Yaskawa INFORM job: DEMO_ROOF_UPPER_0625_3PAINT_33.JBI

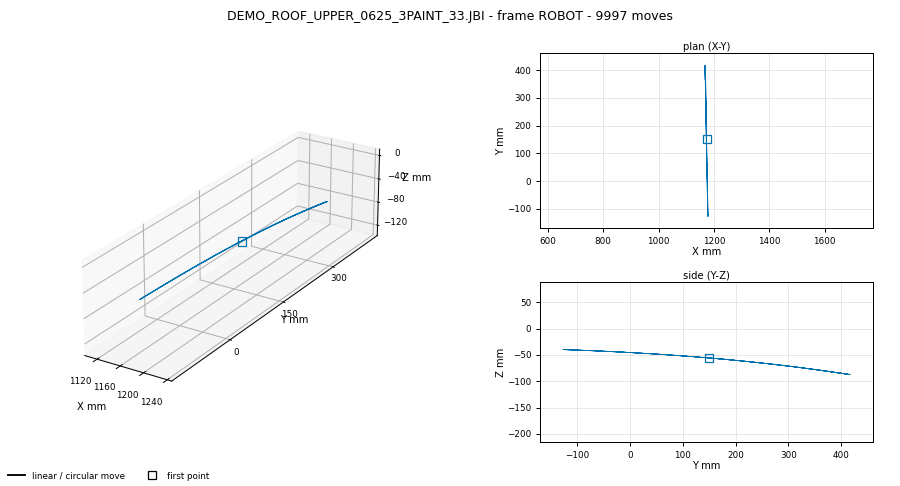
[picture p0: tool path of DEMO_ROOF_UPPER_0625_3PAINT_33.JBI in frame ROBOT, 9997 of 9997 moves have a stored position in this frame; points joined in program order, loops and branches not executed]
/JOB
//NAME DEMO_ROOF_UPPER_0625_3PAINT33
//POS
///NPOS 9997,0,0,0,0,0
///TOOL 0
///USER 0
///POSTYPE ROBOT
///RECTAN
///RCONF 1,0,0,0,0,0,0,0,0,0,0,0,0,0,0,0,0,0,0,0,0,0,0,0
C00000=1173.665,150.338,-55.820,-178.432,6.530,148.733
C00001=1173.661,150.587,-55.840,-178.430,6.532,148.732
C00002=1173.656,150.836,-55.861,-178.427,6.533,148.732
C00003=1173.651,151.085,-55.883,-178.424,6.535,148.732
C00004=1173.646,151.335,-55.904,-178.422,6.536,148.731
C00005=1173.642,151.583,-55.925,-178.420,6.538,148.731
C00006=1173.637,151.832,-55.946,-178.417,6.540,148.730
C00007=1173.632,152.082,-55.967,-178.414,6.541,148.730
C00008=1173.627,152.330,-55.988,-178.411,6.543,148.730
C00009=1173.623,152.580,-56.010,-178.409,6.545,148.729
C00010=1173.618,152.828,-56.031,-178.406,6.547,148.729
C00011=1173.613,153.078,-56.052,-178.403,6.548,148.728
C00012=1173.608,153.327,-56.073,-178.401,6.550,148.728
C00013=1173.604,153.575,-56.094,-178.398,6.552,148.728
C00014=1173.599,153.825,-56.116,-178.395,6.554,148.727
C00015=1173.594,154.074,-56.137,-178.393,6.555,148.727
C00016=1173.590,154.323,-56.158,-178.390,6.557,148.727
C00017=1173.585,154.571,-56.179,-178.387,6.559,148.726
C00018=1173.580,154.821,-56.201,-178.385,6.561,148.726
C00019=1173.575,155.070,-56.223,-178.382,6.562,148.725
C00020=1173.571,155.319,-56.243,-178.379,6.564,148.725
C00021=1173.566,155.568,-56.265,-178.377,6.566,148.725
C00022=1173.562,155.817,-56.287,-178.374,6.568,148.724
C00023=1173.557,156.066,-56.308,-178.371,6.570,148.724
C00024=1173.552,156.315,-56.329,-178.368,6.571,148.724
C00025=1173.547,156.564,-56.350,-178.366,6.573,148.723
C00026=1173.543,156.813,-56.372,-178.363,6.575,148.723
C00027=1173.538,157.062,-56.393,-178.360,6.577,148.722
C00028=1173.533,157.311,-56.414,-178.358,6.578,148.722
C00029=1173.529,157.560,-56.436,-178.355,6.580,148.721
C00030=1173.524,157.810,-56.457,-178.352,6.581,148.721
C00031=1173.519,158.078,-56.481,-178.349,6.583,148.721
C00032=1173.514,158.348,-56.504,-178.346,6.586,148.720
C00033=1173.509,158.617,-56.527,-178.343,6.588,148.720
C00034=1173.504,158.885,-56.551,-178.340,6.589,148.720
C00035=1173.499,159.135,-56.572,-178.338,6.591,148.719
C00036=1173.494,159.383,-56.594,-178.335,6.593,148.719
C00037=1173.489,159.633,-56.616,-178.332,6.595,148.719
C00038=1173.484,159.882,-56.637,-178.330,6.596,148.718
C00039=1173.480,160.130,-56.658,-178.327,6.598,148.718
C00040=1173.476,160.379,-56.680,-178.324,6.600,148.717
C00041=1173.471,160.628,-56.701,-178.322,6.602,148.717
C00042=1173.466,160.877,-56.723,-178.319,6.603,148.717
C00043=1173.462,161.127,-56.745,-178.316,6.605,148.716
C00044=1173.457,161.375,-56.766,-178.314,6.607,148.716
C00045=1173.452,161.625,-56.788,-178.311,6.609,148.716
C00046=1173.448,161.873,-56.810,-178.308,6.610,148.715
C00047=1173.443,162.122,-56.832,-178.306,6.612,148.715
C00048=1173.438,162.371,-56.854,-178.303,6.614,148.714
C00049=1173.433,162.621,-56.875,-178.300,6.616,148.714
C00050=1173.429,162.870,-56.897,-178.297,6.618,148.714
C00051=1173.424,163.119,-56.918,-178.294,6.620,148.713
C00052=1173.419,163.367,-56.940,-178.292,6.622,148.713
C00053=1173.415,163.617,-56.962,-178.289,6.624,148.713
C00054=1173.410,163.865,-56.984,-178.286,6.625,148.712
C00055=1173.405,164.115,-57.006,-178.283,6.627,148.712
C00056=1173.400,164.363,-57.028,-178.281,6.629,148.711
C00057=1173.396,164.613,-57.050,-178.278,6.631,148.711
C00058=1173.391,164.861,-57.072,-178.275,6.632,148.711
C00059=1173.386,165.110,-57.094,-178.273,6.634,148.710
C00060=1173.382,165.359,-57.116,-178.271,6.636,148.710
C00061=1173.377,165.608,-57.137,-178.268,6.638,148.710
C00062=1173.373,165.857,-57.159,-178.265,6.640,148.709
C00063=1173.368,166.106,-57.181,-178.262,6.641,148.709
C00064=1173.364,166.355,-57.203,-178.260,6.643,148.709
C00065=1173.358,166.604,-57.225,-178.257,6.645,148.708
C00066=1173.354,166.854,-57.247,-178.254,6.647,148.708
C00067=1173.349,167.102,-57.269,-178.251,6.649,148.708
C00068=1173.345,167.352,-57.291,-178.248,6.651,148.707
C00069=1173.340,167.600,-57.313,-178.246,6.653,148.707
C00070=1173.335,167.850,-57.335,-178.243,6.655,148.707
C00071=1173.330,168.099,-57.357,-178.240,6.656,148.706
C00072=1173.326,168.348,-57.379,-178.238,6.658,148.706
C00073=1173.321,168.597,-57.401,-178.235,6.660,148.705
C00074=1173.317,168.845,-57.424,-178.232,6.662,148.705
C00075=1173.312,169.094,-57.445,-178.230,6.663,148.705
C00076=1173.307,169.344,-57.468,-178.227,6.666,148.705
C00077=1173.302,169.592,-57.490,-178.225,6.667,148.704
C00078=1173.298,169.842,-57.512,-178.222,6.669,148.704
C00079=1173.293,170.090,-57.534,-178.219,6.671,148.703
C00080=1173.288,170.339,-57.557,-178.216,6.673,148.703
C00081=1173.283,170.588,-57.578,-178.213,6.675,148.703
C00082=1173.279,170.837,-57.600,-178.211,6.677,148.702
C00083=1173.275,171.087,-57.622,-178.208,6.679,148.702
C00084=1173.269,171.335,-57.645,-178.205,6.680,148.702
C00085=1173.265,171.584,-57.667,-178.203,6.682,148.701
C00086=1173.260,171.833,-57.689,-178.200,6.684,148.701
C00087=1173.256,172.082,-57.713,-178.197,6.686,148.701
C00088=1173.251,172.331,-57.734,-178.195,6.688,148.700
C00089=1173.247,172.580,-57.756,-178.192,6.690,148.700
C00090=1173.241,172.830,-57.779,-178.189,6.692,148.700
C00091=1173.237,173.078,-57.801,-178.187,6.694,148.699
C00092=1173.233,173.327,-57.823,-178.184,6.696,148.699
C00093=1173.227,173.575,-57.846,-178.181,6.698,148.699
C00094=1173.223,173.825,-57.868,-178.178,6.699,148.698
C00095=1173.219,174.074,-57.890,-178.176,6.701,148.698
C00096=1173.214,174.322,-57.913,-178.173,6.703,148.698
C00097=1173.209,174.572,-57.935,-178.171,6.705,148.697
C00098=1173.205,174.821,-57.958,-178.168,6.708,148.697
C00099=1173.200,175.069,-57.981,-178.165,6.709,148.697
C00100=1173.195,175.319,-58.003,-178.162,6.711,148.696
C00101=1173.190,175.567,-58.026,-178.160,6.713,148.696
C00102=1173.186,175.816,-58.048,-178.157,6.715,148.696
C00103=1173.181,176.065,-58.071,-178.154,6.716,148.695
C00104=1173.176,176.314,-58.093,-178.152,6.718,148.695
C00105=1173.172,176.563,-58.115,-178.149,6.721,148.695
C00106=1173.167,176.812,-58.138,-178.146,6.723,148.694
C00107=1173.163,177.060,-58.160,-178.143,6.725,148.694
C00108=1173.158,177.310,-58.183,-178.141,6.726,148.694
C00109=1173.154,177.559,-58.206,-178.138,6.728,148.693
C00110=1173.149,177.808,-58.229,-178.135,6.730,148.693
C00111=1173.144,178.056,-58.251,-178.133,6.732,148.693
C00112=1173.140,178.305,-58.274,-178.130,6.735,148.692
C00113=1173.135,178.555,-58.296,-178.127,6.736,148.692
C00114=1173.130,178.803,-58.319,-178.125,6.738,148.692
C00115=1173.126,179.052,-58.341,-178.122,6.740,148.691
C00116=1173.121,179.301,-58.365,-178.119,6.742,148.691
C00117=1173.117,179.550,-58.387,-178.117,6.743,148.691
C00118=1173.111,179.799,-58.410,-178.114,6.745,148.690
C00119=1173.107,180.048,-58.433,-178.111,6.748,148.690
C00120=1173.103,180.297,-58.456,-178.108,6.750,148.690
C00121=1173.098,180.546,-58.478,-178.106,6.752,148.689
C00122=1173.093,180.795,-58.501,-178.103,6.753,148.689
C00123=1173.088,181.044,-58.524,-178.100,6.755,148.689
C00124=1173.084,181.293,-58.546,-178.098,6.757,148.688
C00125=1173.080,181.542,-58.570,-178.095,6.760,148.688
C00126=1173.075,181.790,-58.592,-178.092,6.762,148.688
C00127=1173.070,182.039,-58.615,-178.090,6.764,148.688
C00128=1173.065,182.289,-58.638,-178.087,6.765,148.687
C00129=1173.061,182.537,-58.661,-178.084,6.767,148.687
C00130=1173.056,182.786,-58.684,-178.081,6.770,148.686
C00131=1173.051,183.035,-58.707,-178.079,6.772,148.686
C00132=1173.047,183.284,-58.729,-178.076,6.774,148.686
C00133=1173.042,183.533,-58.753,-178.073,6.775,148.686
C00134=1173.038,183.782,-58.775,-178.071,6.777,148.685
C00135=1173.033,184.052,-58.800,-178.067,6.780,148.685
C00136=1173.028,184.321,-58.825,-178.065,6.781,148.685
C00137=1173.023,184.591,-58.850,-178.062,6.784,148.684
C00138=1173.018,184.860,-58.876,-178.059,6.786,148.684
C00139=1173.013,185.110,-58.898,-178.056,6.788,148.684
C00140=1173.009,185.358,-58.921,-178.053,6.791,148.683
C00141=1173.004,185.607,-58.944,-178.051,6.792,148.683
C00142=1172.999,185.856,-58.967,-178.048,6.794,148.683
C00143=1172.994,186.105,-58.991,-178.045,6.796,148.682
C00144=1172.990,186.353,-59.014,-178.043,6.798,148.682
C00145=1172.986,186.603,-59.037,-178.040,6.801,148.682
C00146=1172.981,186.852,-59.060,-178.037,6.802,148.681
C00147=1172.976,187.101,-59.084,-178.035,6.804,148.681
C00148=1172.972,187.349,-59.106,-178.032,6.806,148.681
C00149=1172.967,187.598,-59.129,-178.030,6.808,148.681
C00150=1172.962,187.847,-59.153,-178.026,6.811,148.680
C00151=1172.958,188.096,-59.176,-178.024,6.812,148.680
C00152=1172.953,188.345,-59.199,-178.021,6.814,148.680
C00153=1172.949,188.593,-59.222,-178.018,6.816,148.679
C00154=1172.944,188.842,-59.246,-178.016,6.819,148.679
C00155=1172.940,189.092,-59.269,-178.013,6.821,148.679
C00156=1172.935,189.341,-59.292,-178.010,6.822,148.678
C00157=1172.930,189.589,-59.315,-178.008,6.824,148.678
C00158=1172.925,189.837,-59.339,-178.005,6.826,148.678
C00159=1172.921,190.086,-59.363,-178.002,6.829,148.678
C00160=1172.917,190.335,-59.385,-177.999,6.831,148.677
C00161=1172.912,190.584,-59.409,-177.997,6.832,148.677
C00162=1172.907,190.833,-59.432,-177.995,6.835,148.677
C00163=1172.903,191.082,-59.456,-177.991,6.837,148.676
C00164=1172.898,191.331,-59.479,-177.989,6.839,148.676
C00165=1172.893,191.580,-59.503,-177.986,6.841,148.676
C00166=1172.889,191.829,-59.526,-177.983,6.842,148.675
C00167=1172.884,192.078,-59.550,-177.981,6.845,148.675
C00168=1172.879,192.327,-59.573,-177.978,6.847,148.675
C00169=1172.875,192.575,-59.597,-177.975,6.849,148.675
C00170=1172.870,192.824,-59.620,-177.973,6.851,148.674
C00171=1172.866,193.073,-59.644,-177.970,6.854,148.674
C00172=1172.861,193.322,-59.667,-177.967,6.855,148.674
C00173=1172.856,193.571,-59.691,-177.964,6.857,148.673
C00174=1172.852,193.820,-59.715,-177.962,6.859,148.673
C00175=1172.847,194.069,-59.738,-177.959,6.862,148.673
C00176=1172.843,194.317,-59.762,-177.956,6.864,148.673
C00177=1172.838,194.566,-59.785,-177.954,6.866,148.672
C00178=1172.833,194.815,-59.809,-177.951,6.868,148.672
C00179=1172.829,195.064,-59.833,-177.948,6.870,148.672
C00180=1172.824,195.313,-59.856,-177.946,6.872,148.671
C00181=1172.819,195.562,-59.880,-177.943,6.874,148.671
C00182=1172.815,195.810,-59.904,-177.940,6.877,148.671
C00183=1172.810,196.059,-59.927,-177.937,6.879,148.671
C00184=1172.806,196.307,-59.951,-177.935,6.880,148.670
C00185=1172.801,196.557,-59.974,-177.933,6.882,148.670
C00186=1172.797,196.806,-59.998,-177.929,6.885,148.670
C00187=1172.792,197.054,-60.022,-177.927,6.887,148.669
C00188=1172.787,197.303,-60.045,-177.924,6.889,148.669
C00189=1172.784,197.552,-60.070,-177.921,6.892,148.669
C00190=1172.779,197.801,-60.093,-177.918,6.893,148.669
C00191=1172.775,198.050,-60.117,-177.916,6.895,148.668
C00192=1172.769,198.299,-60.141,-177.914,6.897,148.668
C00193=1172.765,198.547,-60.165,-177.910,6.900,148.668
C00194=1172.760,198.796,-60.188,-177.908,6.902,148.668
C00195=1172.756,199.045,-60.213,-177.905,6.903,148.667
C00196=1172.751,199.294,-60.236,-177.902,6.906,148.667
C00197=1172.747,199.542,-60.260,-177.900,6.908,148.667
C00198=1172.742,199.791,-60.284,-177.897,6.910,148.666
C00199=1172.737,200.041,-60.308,-177.894,6.913,148.666
C00200=1172.733,200.289,-60.332,-177.891,6.915,148.666
C00201=1172.728,200.538,-60.356,-177.889,6.916,148.666
C00202=1172.724,200.787,-60.380,-177.887,6.919,148.665
C00203=1172.719,201.035,-60.404,-177.883,6.921,148.665
C00204=1172.714,201.284,-60.428,-177.881,6.923,148.665
C00205=1172.710,201.533,-60.452,-177.879,6.925,148.665
C00206=1172.706,201.782,-60.476,-177.875,6.928,148.664
C00207=1172.701,202.031,-60.500,-177.873,6.929,148.664
C00208=1172.697,202.279,-60.524,-177.870,6.932,148.664
C00209=1172.692,202.528,-60.549,-177.867,6.934,148.664
C00210=1172.687,202.776,-60.573,-177.864,6.936,148.663
C00211=1172.683,203.026,-60.596,-177.862,6.938,148.663
C00212=1172.678,203.275,-60.621,-177.859,6.941,148.663
C00213=1172.674,203.523,-60.645,-177.856,6.942,148.662
C00214=1172.669,203.772,-60.669,-177.854,6.945,148.662
C00215=1172.664,204.021,-60.693,-177.851,6.947,148.662
C00216=1172.660,204.270,-60.718,-177.848,6.949,148.662
C00217=1172.656,204.519,-60.742,-177.846,6.951,148.662
C00218=1172.651,204.767,-60.766,-177.843,6.954,148.661
C00219=1172.646,205.016,-60.790,-177.840,6.955,148.661
C00220=1172.642,205.265,-60.814,-177.838,6.958,148.661
C00221=1172.638,205.514,-60.838,-177.835,6.960,148.660
C00222=1172.632,205.763,-60.863,-177.832,6.962,148.660
C00223=1172.628,206.011,-60.887,-177.830,6.964,148.660
C00224=1172.623,206.260,-60.912,-177.827,6.967,148.660
C00225=1172.619,206.509,-60.936,-177.824,6.969,148.660
C00226=1172.615,206.757,-60.960,-177.822,6.971,148.659
C00227=1172.610,207.006,-60.985,-177.819,6.973,148.659
C00228=1172.606,207.255,-61.009,-177.816,6.975,148.659
C00229=1172.601,207.504,-61.034,-177.813,6.978,148.658
C00230=1172.596,207.753,-61.057,-177.810,6.980,148.658
C00231=1172.592,208.001,-61.081,-177.808,6.982,148.658
C00232=1172.587,208.251,-61.106,-177.805,6.984,148.658
C00233=1172.583,208.499,-61.130,-177.803,6.987,148.658
C00234=1172.577,208.748,-61.155,-177.800,6.988,148.657
C00235=1172.574,208.997,-61.180,-177.797,6.991,148.657
C00236=1172.569,209.246,-61.204,-177.795,6.993,148.657
C00237=1172.564,209.493,-61.229,-177.792,6.995,148.656
C00238=1172.559,209.742,-61.254,-177.789,6.998,148.656
C00239=1172.554,210.014,-61.280,-177.786,7.000,148.656
C00240=1172.549,210.284,-61.307,-177.783,7.002,148.656
C00241=1172.545,210.554,-61.333,-177.780,7.005,148.655
C00242=1172.540,210.824,-61.360,-177.777,7.007,148.655
C00243=1172.535,211.073,-61.385,-177.775,7.010,148.655
C00244=1172.531,211.322,-61.409,-177.772,7.011,148.655
C00245=1172.526,211.571,-61.434,-177.769,7.014,148.654
C00246=1172.521,211.819,-61.459,-177.767,7.016,148.654
C00247=1172.518,212.068,-61.484,-177.764,7.018,148.654
C00248=1172.513,212.317,-61.508,-177.761,7.021,148.654
C00249=1172.508,212.565,-61.532,-177.759,7.023,148.653
C00250=1172.504,212.815,-61.557,-177.756,7.026,148.653
C00251=1172.500,213.063,-61.582,-177.753,7.027,148.653
C00252=1172.495,213.312,-61.607,-177.751,7.029,148.653
C00253=1172.490,213.561,-61.632,-177.748,7.032,148.652
C00254=1172.485,213.809,-61.656,-177.745,7.034,148.652
C00255=1172.481,214.058,-61.682,-177.742,7.037,148.652
C00256=1172.476,214.307,-61.706,-177.740,7.039,148.652
C00257=1172.472,214.556,-61.731,-177.737,7.042,148.652
C00258=1172.467,214.805,-61.755,-177.734,7.043,148.651
C00259=1172.463,215.052,-61.780,-177.732,7.046,148.651
C00260=1172.459,215.302,-61.805,-177.729,7.048,148.651
C00261=1172.453,215.550,-61.830,-177.726,7.050,148.651
C00262=1172.449,215.799,-61.856,-177.723,7.053,148.650
C00263=1172.445,216.048,-61.880,-177.721,7.055,148.650
C00264=1172.441,216.297,-61.905,-177.718,7.057,148.650
C00265=1172.435,216.545,-61.930,-177.715,7.059,148.650
C00266=1172.432,216.794,-61.955,-177.713,7.062,148.650
C00267=1172.427,217.042,-61.980,-177.710,7.064,148.649
C00268=1172.422,217.292,-62.005,-177.708,7.066,148.649
C00269=1172.418,217.540,-62.030,-177.704,7.069,148.649
C00270=1172.414,217.789,-62.055,-177.702,7.071,148.648
C00271=1172.409,218.038,-62.080,-177.700,7.073,148.648
C00272=1172.404,218.287,-62.105,-177.696,7.075,148.648
C00273=1172.400,218.535,-62.129,-177.694,7.078,148.648
C00274=1172.396,218.784,-62.155,-177.691,7.080,148.648
C00275=1172.391,219.033,-62.180,-177.689,7.082,148.648
C00276=1172.386,219.281,-62.206,-177.685,7.085,148.647
C00277=1172.382,219.529,-62.231,-177.683,7.087,148.647
C00278=1172.378,219.779,-62.255,-177.680,7.090,148.647
C00279=1172.373,220.027,-62.281,-177.678,7.092,148.647
C00280=1172.368,220.276,-62.306,-177.675,7.094,148.646
C00281=1172.364,220.524,-62.331,-177.672,7.097,148.646
C00282=1172.359,220.774,-62.356,-177.670,7.098,148.646
C00283=1172.354,221.022,-62.382,-177.667,7.101,148.646
C00284=1172.351,221.270,-62.407,-177.664,7.103,148.646
C00285=1172.346,221.519,-62.431,-177.662,7.106,148.645
C00286=1172.341,221.768,-62.457,-177.659,7.108,148.645
C00287=1172.337,222.017,-62.483,-177.656,7.111,148.645
C00288=1172.332,222.265,-62.508,-177.653,7.113,148.645
C00289=1172.328,222.514,-62.533,-177.651,7.115,148.645
C00290=1172.323,222.762,-62.559,-177.648,7.117,148.644
C00291=1172.318,223.012,-62.584,-177.645,7.120,148.644
C00292=1172.314,223.260,-62.609,-177.643,7.122,148.644
C00293=1172.309,223.509,-62.635,-177.640,7.124,148.644
C00294=1172.306,223.758,-62.659,-177.637,7.127,148.643
C00295=1172.301,224.006,-62.685,-177.635,7.129,148.643
C00296=1172.297,224.255,-62.710,-177.632,7.132,148.643
C00297=1172.292,224.503,-62.736,-177.630,7.134,148.643
C00298=1172.288,224.751,-62.762,-177.626,7.136,148.643
C00299=1172.283,225.001,-62.787,-177.624,7.138,148.642
C00300=1172.278,225.249,-62.812,-177.621,7.141,148.642
C00301=1172.274,225.498,-62.838,-177.619,7.143,148.642
C00302=1172.270,225.747,-62.863,-177.616,7.146,148.642
C00303=1172.265,225.995,-62.889,-177.613,7.148,148.642
C00304=1172.261,226.244,-62.915,-177.610,7.151,148.641
C00305=1172.256,226.493,-62.940,-177.608,7.153,148.641
C00306=1172.251,226.741,-62.965,-177.605,7.155,148.641
C00307=1172.247,226.990,-62.991,-177.603,7.157,148.641
C00308=1172.243,227.239,-63.017,-177.599,7.160,148.641
C00309=1172.237,227.487,-63.043,-177.597,7.162,148.640
C00310=1172.233,227.736,-63.068,-177.594,7.165,148.640
C00311=1172.229,227.985,-63.094,-177.592,7.167,148.640
C00312=1172.224,228.233,-63.119,-177.589,7.170,148.640
C00313=1172.220,228.482,-63.145,-177.586,7.172,148.640
C00314=1172.216,228.730,-63.171,-177.584,7.175,148.640
C00315=1172.211,228.978,-63.196,-177.581,7.176,148.639
C00316=1172.206,229.227,-63.222,-177.578,7.179,148.639
C00317=1172.202,229.476,-63.248,-177.576,7.182,148.639
C00318=1172.198,229.725,-63.274,-177.573,7.184,148.639
C00319=1172.192,229.973,-63.300,-177.570,7.186,148.639
C00320=1172.188,230.222,-63.325,-177.567,7.189,148.638
C00321=1172.184,230.471,-63.351,-177.565,7.192,148.638
C00322=1172.180,230.720,-63.377,-177.562,7.194,148.638
C00323=1172.175,230.968,-63.402,-177.559,7.197,148.638
C00324=1172.171,231.217,-63.428,-177.557,7.199,148.638
C00325=1172.166,231.465,-63.455,-177.554,7.201,148.637
C00326=1172.162,231.714,-63.481,-177.551,7.203,148.637
C00327=1172.157,231.962,-63.506,-177.548,7.206,148.637
C00328=1172.153,232.211,-63.532,-177.546,7.208,148.637
C00329=1172.149,232.460,-63.558,-177.543,7.211,148.637
C00330=1172.144,232.709,-63.584,-177.541,7.213,148.637
C00331=1172.139,232.958,-63.610,-177.538,7.216,148.636
C00332=1172.135,233.205,-63.636,-177.535,7.218,148.636
C00333=1172.131,233.454,-63.662,-177.533,7.221,148.636
C00334=1172.126,233.703,-63.688,-177.530,7.224,148.636
C00335=1172.121,233.952,-63.714,-177.527,7.225,148.636
C00336=1172.118,234.200,-63.740,-177.524,7.228,148.636
C00337=1172.112,234.448,-63.766,-177.522,7.230,148.635
C00338=1172.108,234.697,-63.792,-177.519,7.233,148.635
C00339=1172.104,234.945,-63.818,-177.517,7.235,148.635
C00340=1172.100,235.194,-63.844,-177.514,7.238,148.635
C00341=1172.095,235.443,-63.870,-177.511,7.240,148.635
C00342=1172.090,235.692,-63.896,-177.509,7.243,148.635
C00343=1172.085,235.963,-63.925,-177.505,7.246,148.634
C00344=1172.080,236.234,-63.954,-177.503,7.249,148.634
C00345=1172.076,236.506,-63.982,-177.499,7.251,148.634
C00346=1172.071,236.778,-64.011,-177.497,7.254,148.634
C00347=1172.066,237.027,-64.037,-177.494,7.256,148.634
C00348=1172.062,237.275,-64.063,-177.491,7.259,148.633
C00349=1172.057,237.524,-64.090,-177.489,7.261,148.633
C00350=1172.053,237.773,-64.116,-177.486,7.264,148.633
C00351=1172.049,238.021,-64.142,-177.484,7.266,148.633
C00352=1172.044,238.269,-64.168,-177.480,7.268,148.633
C00353=1172.040,238.517,-64.195,-177.478,7.271,148.633
C00354=1172.035,238.767,-64.221,-177.475,7.274,148.632
C00355=1172.031,239.015,-64.247,-177.472,7.276,148.632
C00356=1172.026,239.264,-64.274,-177.470,7.278,148.632
C00357=1172.022,239.512,-64.300,-177.467,7.281,148.632
C00358=1172.017,239.761,-64.327,-177.464,7.284,148.632
C00359=1172.013,240.009,-64.353,-177.462,7.286,148.632
C00360=1172.008,240.258,-64.379,-177.459,7.289,148.632
C00361=1172.004,240.507,-64.406,-177.457,7.291,148.631
C00362=1171.999,240.756,-64.432,-177.454,7.294,148.631
C00363=1171.995,241.004,-64.459,-177.451,7.297,148.631
C00364=1171.991,241.252,-64.486,-177.449,7.299,148.631
C00365=1171.986,241.501,-64.511,-177.446,7.301,148.631
C00366=1171.982,241.750,-64.538,-177.443,7.304,148.631
C00367=1171.978,241.998,-64.565,-177.441,7.307,148.631
C00368=1171.972,242.246,-64.591,-177.437,7.309,148.630
C00369=1171.968,242.495,-64.617,-177.435,7.311,148.630
C00370=1171.964,242.743,-64.644,-177.432,7.314,148.630
C00371=1171.960,242.992,-64.670,-177.430,7.317,148.630
C00372=1171.955,243.240,-64.697,-177.427,7.319,148.630
C00373=1171.950,243.489,-64.724,-177.424,7.322,148.630
C00374=1171.946,243.737,-64.751,-177.422,7.324,148.630
C00375=1171.942,243.987,-64.778,-177.419,7.327,148.629
C00376=1171.938,244.235,-64.804,-177.416,7.330,148.629
C00377=1171.933,244.484,-64.831,-177.414,7.332,148.629
C00378=1171.929,244.732,-64.858,-177.411,7.335,148.629
C00379=1171.925,244.981,-64.884,-177.408,7.337,148.629
C00380=1171.920,245.229,-64.911,-177.406,7.340,148.629
C00381=1171.915,245.478,-64.938,-177.403,7.343,148.629
C00382=1171.911,245.726,-64.964,-177.401,7.345,148.628
C00383=1171.907,245.974,-64.991,-177.398,7.347,148.628
C00384=1171.902,246.223,-65.019,-177.395,7.350,148.628
C00385=1171.898,246.472,-65.044,-177.393,7.352,148.628
C00386=1171.893,246.720,-65.071,-177.390,7.355,148.628
C00387=1171.888,246.969,-65.098,-177.387,7.358,148.628
C00388=1171.885,247.217,-65.125,-177.385,7.360,148.628
C00389=1171.880,247.465,-65.152,-177.382,7.363,148.627
C00390=1171.875,247.714,-65.179,-177.379,7.366,148.627
C00391=1171.871,247.962,-65.206,-177.376,7.368,148.627
C00392=1171.867,248.211,-65.233,-177.374,7.371,148.627
C00393=1171.863,248.460,-65.260,-177.371,7.374,148.627
C00394=1171.858,248.708,-65.287,-177.369,7.376,148.627
C00395=1171.853,248.957,-65.314,-177.366,7.379,148.627
C00396=1171.849,249.205,-65.341,-177.363,7.382,148.627
C00397=1171.845,249.454,-65.368,-177.361,7.384,148.626
C00398=1171.840,249.702,-65.395,-177.358,7.387,148.626
C00399=1171.835,249.950,-65.422,-177.355,7.390,148.626
C00400=1171.831,250.200,-65.449,-177.352,7.391,148.626
C00401=1171.827,250.448,-65.476,-177.350,7.394,148.626
C00402=1171.823,250.696,-65.503,-177.347,7.397,148.626
C00403=1171.818,250.945,-65.530,-177.345,7.400,148.626
C00404=1171.814,251.193,-65.558,-177.342,7.402,148.626
C00405=1171.809,251.441,-65.585,-177.339,7.405,148.625
C00406=1171.804,251.690,-65.612,-177.337,7.407,148.625
C00407=1171.801,251.939,-65.638,-177.334,7.410,148.625
C00408=1171.796,252.187,-65.666,-177.331,7.413,148.625
C00409=1171.792,252.436,-65.693,-177.329,7.415,148.625
C00410=1171.787,252.683,-65.720,-177.326,7.418,148.625
C00411=1171.783,252.932,-65.747,-177.323,7.421,148.625
C00412=1171.779,253.181,-65.775,-177.321,7.423,148.625
C00413=1171.774,253.430,-65.802,-177.318,7.426,148.625
C00414=1171.769,253.678,-65.829,-177.315,7.429,148.625
C00415=1171.765,253.926,-65.857,-177.313,7.431,148.624
C00416=1171.761,254.175,-65.884,-177.310,7.434,148.624
C00417=1171.756,254.424,-65.911,-177.307,7.437,148.624
C00418=1171.752,254.672,-65.939,-177.304,7.440,148.624
C00419=1171.747,254.920,-65.966,-177.302,7.442,148.624
C00420=1171.743,255.168,-65.993,-177.299,7.445,148.624
C00421=1171.740,255.417,-66.021,-177.297,7.448,148.624
C00422=1171.735,255.665,-66.048,-177.294,7.450,148.624
C00423=1171.730,255.914,-66.075,-177.291,7.453,148.623
C00424=1171.726,256.162,-66.103,-177.289,7.455,148.623
C00425=1171.721,256.411,-66.131,-177.286,7.458,148.623
C00426=1171.717,256.660,-66.158,-177.284,7.461,148.623
C00427=1171.712,256.908,-66.185,-177.281,7.464,148.623
C00428=1171.708,257.157,-66.213,-177.278,7.467,148.623
C00429=1171.704,257.405,-66.241,-177.275,7.468,148.623
C00430=1171.699,257.653,-66.268,-177.273,7.471,148.623
C00431=1171.695,257.901,-66.296,-177.270,7.474,148.623
C00432=1171.691,258.150,-66.323,-177.267,7.477,148.623
C00433=1171.686,258.398,-66.351,-177.265,7.479,148.623
C00434=1171.682,258.647,-66.378,-177.262,7.482,148.623
C00435=1171.678,258.895,-66.406,-177.260,7.485,148.622
C00436=1171.673,259.144,-66.433,-177.257,7.487,148.622
C00437=1171.669,259.392,-66.461,-177.254,7.490,148.622
C00438=1171.664,259.641,-66.489,-177.251,7.493,148.622
C00439=1171.660,259.889,-66.517,-177.249,7.496,148.622
C00440=1171.655,260.137,-66.544,-177.246,7.498,148.622
C00441=1171.651,260.386,-66.572,-177.244,7.501,148.622
C00442=1171.647,260.634,-66.600,-177.241,7.504,148.622
C00443=1171.642,260.882,-66.627,-177.238,7.507,148.622
C00444=1171.639,261.131,-66.655,-177.236,7.509,148.622
C00445=1171.633,261.380,-66.682,-177.233,7.512,148.622
C00446=1171.630,261.628,-66.711,-177.231,7.515,148.622
C00447=1171.624,261.901,-66.741,-177.227,7.518,148.621
C00448=1171.620,262.174,-66.772,-177.225,7.521,148.621
C00449=1171.615,262.448,-66.802,-177.222,7.524,148.621
C00450=1171.610,262.720,-66.833,-177.219,7.527,148.621
C00451=1171.606,262.969,-66.861,-177.216,7.530,148.621
C00452=1171.602,263.217,-66.888,-177.214,7.533,148.621
C00453=1171.598,263.465,-66.917,-177.211,7.536,148.621
C00454=1171.592,263.714,-66.944,-177.209,7.538,148.621
C00455=1171.588,263.962,-66.972,-177.206,7.541,148.621
C00456=1171.584,264.211,-67.000,-177.203,7.543,148.621
C00457=1171.579,264.459,-67.029,-177.200,7.546,148.620
C00458=1171.575,264.708,-67.056,-177.198,7.548,148.620
C00459=1171.571,264.956,-67.084,-177.195,7.551,148.620
C00460=1171.566,265.205,-67.112,-177.192,7.554,148.620
C00461=1171.562,265.453,-67.140,-177.190,7.557,148.620
C00462=1171.558,265.701,-67.168,-177.187,7.560,148.620
C00463=1171.553,265.949,-67.197,-177.185,7.562,148.620
C00464=1171.549,266.197,-67.225,-177.182,7.565,148.620
C00465=1171.545,266.446,-67.253,-177.179,7.568,148.620
C00466=1171.540,266.695,-67.280,-177.176,7.571,148.620
C00467=1171.536,266.943,-67.308,-177.174,7.573,148.620
C00468=1171.532,267.191,-67.336,-177.171,7.576,148.620
C00469=1171.527,267.440,-67.365,-177.169,7.579,148.620
C00470=1171.523,267.688,-67.393,-177.166,7.582,148.620
C00471=1171.518,267.937,-67.422,-177.163,7.585,148.620
C00472=1171.514,268.185,-67.449,-177.161,7.587,148.620
C00473=1171.510,268.433,-67.477,-177.158,7.590,148.620
C00474=1171.505,268.681,-67.506,-177.156,7.593,148.619
C00475=1171.501,268.930,-67.534,-177.153,7.596,148.619
C00476=1171.497,269.179,-67.563,-177.151,7.599,148.619
C00477=1171.492,269.427,-67.590,-177.148,7.602,148.619
C00478=1171.488,269.676,-67.619,-177.145,7.604,148.619
C00479=1171.484,269.923,-67.648,-177.142,7.607,148.619
C00480=1171.479,270.172,-67.676,-177.140,7.610,148.619
C00481=1171.475,270.420,-67.704,-177.137,7.613,148.619
C00482=1171.471,270.668,-67.733,-177.135,7.616,148.619
C00483=1171.466,270.916,-67.761,-177.132,7.619,148.619
C00484=1171.462,271.165,-67.789,-177.129,7.621,148.619
C00485=1171.458,271.414,-67.818,-177.127,7.624,148.619
C00486=1171.453,271.661,-67.847,-177.124,7.627,148.619
C00487=1171.449,271.910,-67.875,-177.122,7.630,148.619
C00488=1171.444,272.158,-67.903,-177.119,7.633,148.619
C00489=1171.441,272.407,-67.931,-177.116,7.635,148.619
C00490=1171.436,272.656,-67.960,-177.113,7.638,148.619
C00491=1171.431,272.903,-67.989,-177.111,7.641,148.619
C00492=1171.428,273.152,-68.017,-177.108,7.644,148.618
C00493=1171.423,273.400,-68.046,-177.106,7.647,148.618
C00494=1171.419,273.649,-68.074,-177.103,7.650,148.618
C00495=1171.415,273.897,-68.103,-177.100,7.652,148.618
C00496=1171.409,274.145,-68.132,-177.097,7.655,148.618
C00497=1171.406,274.394,-68.160,-177.095,7.658,148.618
C00498=1171.402,274.642,-68.189,-177.093,7.661,148.618
C00499=1171.397,274.890,-68.217,-177.090,7.664,148.618
C00500=1171.393,275.139,-68.246,-177.088,7.667,148.618
C00501=1171.389,275.387,-68.275,-177.085,7.670,148.618
C00502=1171.384,275.635,-68.303,-177.082,7.673,148.618
C00503=1171.380,275.883,-68.332,-177.080,7.675,148.618
C00504=1171.376,276.132,-68.361,-177.077,7.678,148.618
C00505=1171.370,276.380,-68.390,-177.074,7.681,148.618
C00506=1171.367,276.628,-68.418,-177.072,7.684,148.618
C00507=1171.362,276.877,-68.447,-177.069,7.687,148.618
C00508=1171.358,277.124,-68.476,-177.066,7.690,148.618
C00509=1171.354,277.373,-68.504,-177.063,7.693,148.618
C00510=1171.350,277.621,-68.534,-177.061,7.695,148.618
C00511=1171.345,277.870,-68.562,-177.058,7.698,148.618
C00512=1171.341,278.118,-68.592,-177.056,7.701,148.618
C00513=1171.337,278.366,-68.620,-177.053,7.704,148.618
C00514=1171.333,278.615,-68.649,-177.051,7.707,148.618
C00515=1171.327,278.863,-68.678,-177.048,7.710,148.618
C00516=1171.323,279.111,-68.707,-177.046,7.712,148.618
C00517=1171.320,279.359,-68.736,-177.043,7.715,148.618
C00518=1171.315,279.608,-68.765,-177.040,7.718,148.618
C00519=1171.311,279.855,-68.794,-177.038,7.721,148.618
C00520=1171.306,280.104,-68.823,-177.035,7.724,148.618
C00521=1171.302,280.353,-68.852,-177.032,7.727,148.617
C00522=1171.298,280.601,-68.881,-177.030,7.730,148.618
C00523=1171.293,280.849,-68.909,-177.028,7.733,148.618
C00524=1171.289,281.097,-68.939,-177.025,7.736,148.618
C00525=1171.285,281.345,-68.968,-177.022,7.738,148.617
C00526=1171.281,281.594,-68.997,-177.019,7.741,148.617
C00527=1171.276,281.842,-69.026,-177.017,7.744,148.617
C00528=1171.272,282.090,-69.055,-177.014,7.747,148.617
C00529=1171.267,282.338,-69.085,-177.011,7.750,148.617
C00530=1171.263,282.587,-69.114,-177.009,7.754,148.618
C00531=1171.259,282.835,-69.142,-177.007,7.756,148.617
C00532=1171.255,283.083,-69.172,-177.004,7.759,148.617
C00533=1171.251,283.331,-69.201,-177.001,7.762,148.617
C00534=1171.246,283.580,-69.230,-176.998,7.765,148.617
C00535=1171.242,283.828,-69.259,-176.996,7.768,148.617
C00536=1171.238,284.076,-69.289,-176.993,7.771,148.617
C00537=1171.233,284.325,-69.318,-176.991,7.774,148.617
C00538=1171.229,284.573,-69.348,-176.988,7.777,148.617
C00539=1171.225,284.821,-69.377,-176.985,7.780,148.617
C00540=1171.220,285.069,-69.406,-176.983,7.782,148.617
C00541=1171.216,285.318,-69.435,-176.980,7.785,148.617
C00542=1171.212,285.566,-69.464,-176.978,7.788,148.617
C00543=1171.207,285.814,-69.494,-176.975,7.791,148.617
C00544=1171.203,286.062,-69.523,-176.973,7.794,148.617
C00545=1171.199,286.311,-69.553,-176.970,7.797,148.617
C00546=1171.195,286.559,-69.582,-176.967,7.800,148.617
C00547=1171.191,286.807,-69.612,-176.964,7.803,148.617
C00548=1171.186,287.055,-69.641,-176.962,7.806,148.617
C00549=1171.182,287.303,-69.670,-176.960,7.809,148.617
C00550=1171.177,287.552,-69.700,-176.957,7.812,148.617
C00551=1171.173,287.826,-69.733,-176.954,7.815,148.617
C00552=1171.168,288.102,-69.765,-176.951,7.818,148.617
C00553=1171.163,288.377,-69.798,-176.948,7.821,148.617
C00554=1171.159,288.651,-69.830,-176.945,7.825,148.617
C00555=1171.154,288.899,-69.860,-176.942,7.828,148.617
C00556=1171.149,289.147,-69.890,-176.941,7.831,148.617
C00557=1171.145,289.396,-69.919,-176.938,7.834,148.617
C00558=1171.141,289.644,-69.949,-176.935,7.837,148.617
C00559=1171.137,289.892,-69.979,-176.932,7.840,148.617
C00560=1171.133,290.140,-70.008,-176.930,7.843,148.617
C00561=1171.129,290.388,-70.038,-176.927,7.846,148.617
C00562=1171.124,290.637,-70.068,-176.925,7.849,148.617
C00563=1171.120,290.885,-70.097,-176.922,7.852,148.617
C00564=1171.116,291.133,-70.127,-176.919,7.855,148.617
C00565=1171.112,291.381,-70.157,-176.917,7.858,148.617
C00566=1171.108,291.629,-70.186,-176.914,7.861,148.617
C00567=1171.103,291.878,-70.217,-176.911,7.864,148.617
C00568=1171.098,292.126,-70.246,-176.909,7.866,148.617
C00569=1171.095,292.374,-70.276,-176.906,7.869,148.617
C00570=1171.090,292.622,-70.306,-176.904,7.872,148.617
C00571=1171.085,292.871,-70.336,-176.901,7.875,148.617
C00572=1171.082,293.118,-70.366,-176.899,7.878,148.617
C00573=1171.077,293.366,-70.395,-176.896,7.881,148.617
C00574=1171.073,293.615,-70.425,-176.894,7.885,148.618
C00575=1171.069,293.863,-70.455,-176.891,7.888,148.618
C00576=1171.064,294.111,-70.485,-176.888,7.891,148.617
C00577=1171.060,294.359,-70.514,-176.885,7.894,148.617
C00578=1171.056,294.607,-70.545,-176.883,7.897,148.618
C00579=1171.052,294.856,-70.575,-176.880,7.900,148.618
C00580=1171.048,295.104,-70.605,-176.878,7.903,148.618
C00581=1171.043,295.352,-70.635,-176.875,7.906,148.618
C00582=1171.039,295.601,-70.665,-176.873,7.909,148.618
C00583=1171.035,295.848,-70.695,-176.870,7.912,148.618
C00584=1171.030,296.097,-70.725,-176.868,7.914,148.618
C00585=1171.026,296.345,-70.755,-176.865,7.918,148.618
C00586=1171.022,296.593,-70.784,-176.863,7.920,148.618
C00587=1171.018,296.841,-70.815,-176.860,7.923,148.618
C00588=1171.013,297.089,-70.845,-176.857,7.926,148.618
C00589=1171.009,297.338,-70.876,-176.855,7.930,148.618
C00590=1171.006,297.585,-70.906,-176.852,7.933,148.618
C00591=1171.001,297.834,-70.935,-176.849,7.936,148.618
C00592=1170.997,298.082,-70.966,-176.847,7.939,148.618
C00593=1170.993,298.330,-70.996,-176.844,7.942,148.618
C00594=1170.988,298.578,-71.026,-176.842,7.945,148.618
C00595=1170.984,298.826,-71.056,-176.839,7.948,148.618
C00596=1170.980,299.075,-71.087,-176.837,7.951,148.618
C00597=1170.976,299.322,-71.117,-176.834,7.954,148.618
C00598=1170.971,299.571,-71.147,-176.831,7.957,148.618
C00599=1170.967,299.819,-71.177,-176.829,7.960,148.618
C00600=1170.962,300.067,-71.208,-176.826,7.963,148.618
C00601=1170.958,300.315,-71.238,-176.823,7.966,148.618
C00602=1170.954,300.563,-71.269,-176.821,7.970,148.618
C00603=1170.950,300.811,-71.299,-176.818,7.973,148.618
C00604=1170.946,301.059,-71.330,-176.816,7.976,148.618
C00605=1170.942,301.307,-71.359,-176.813,7.979,148.619
C00606=1170.937,301.555,-71.390,-176.811,7.982,148.619
C00607=1170.934,301.804,-71.420,-176.808,7.985,148.618
C00608=1170.929,302.052,-71.451,-176.806,7.988,148.619
C00609=1170.924,302.300,-71.482,-176.803,7.991,148.619
C00610=1170.920,302.548,-71.511,-176.800,7.994,148.619
C00611=1170.916,302.796,-71.542,-176.798,7.997,148.619
C00612=1170.912,303.044,-71.573,-176.795,8.000,148.619
C00613=1170.908,303.292,-71.603,-176.792,8.003,148.619
C00614=1170.903,303.540,-71.634,-176.790,8.007,148.619
C00615=1170.899,303.788,-71.664,-176.787,8.010,148.619
C00616=1170.895,304.036,-71.696,-176.786,8.012,148.619
C00617=1170.890,304.285,-71.726,-176.783,8.015,148.619
C00618=1170.887,304.533,-71.756,-176.780,8.018,148.619
C00619=1170.882,304.781,-71.787,-176.778,8.021,148.619
C00620=1170.878,305.029,-71.818,-176.775,8.024,148.619
C00621=1170.874,305.277,-71.848,-176.772,8.027,148.619
C00622=1170.869,305.525,-71.879,-176.770,8.031,148.619
C00623=1170.865,305.773,-71.909,-176.767,8.034,148.619
C00624=1170.861,306.021,-71.940,-176.765,8.037,148.620
C00625=1170.857,306.269,-71.971,-176.762,8.040,148.619
C00626=1170.852,306.517,-72.001,-176.760,8.043,148.619
C00627=1170.848,306.766,-72.033,-176.757,8.046,148.620
C00628=1170.844,307.014,-72.063,-176.755,8.049,148.620
C00629=1170.840,307.261,-72.093,-176.752,8.052,148.620
C00630=1170.836,307.510,-72.125,-176.750,8.055,148.620
C00631=1170.831,307.757,-72.156,-176.747,8.058,148.620
C00632=1170.827,308.005,-72.187,-176.745,8.062,148.620
C00633=1170.824,308.254,-72.217,-176.742,8.065,148.620
C00634=1170.819,308.502,-72.248,-176.739,8.069,148.620
C00635=1170.814,308.750,-72.279,-176.736,8.072,148.620
C00636=1170.810,308.998,-72.310,-176.734,8.075,148.620
C00637=1170.806,309.246,-72.341,-176.731,8.078,148.620
C00638=1170.801,309.493,-72.372,-176.729,8.081,148.620
C00639=1170.798,309.742,-72.403,-176.726,8.084,148.621
C00640=1170.794,309.990,-72.434,-176.724,8.087,148.620
C00641=1170.790,310.238,-72.465,-176.721,8.090,148.620
C00642=1170.785,310.486,-72.496,-176.719,8.094,148.621
C00643=1170.781,310.734,-72.527,-176.716,8.097,148.621
C00644=1170.777,310.982,-72.558,-176.714,8.100,148.621
C00645=1170.772,311.230,-72.589,-176.711,8.103,148.621
C00646=1170.769,311.478,-72.620,-176.708,8.106,148.621
C00647=1170.764,311.726,-72.651,-176.706,8.109,148.621
C00648=1170.760,311.974,-72.682,-176.703,8.112,148.621
C00649=1170.756,312.222,-72.713,-176.701,8.115,148.621
C00650=1170.751,312.470,-72.744,-176.698,8.118,148.621
C00651=1170.747,312.719,-72.775,-176.696,8.122,148.621
C00652=1170.743,312.966,-72.807,-176.693,8.125,148.621
C00653=1170.739,313.215,-72.838,-176.691,8.128,148.622
C00654=1170.735,313.462,-72.869,-176.688,8.131,148.622
C00655=1170.730,313.739,-72.904,-176.686,8.134,148.622
C00656=1170.725,314.016,-72.939,-176.682,8.138,148.622
C00657=1170.721,314.293,-72.974,-176.680,8.142,148.622
C00658=1170.716,314.570,-73.009,-176.677,8.145,148.622
C00659=1170.712,314.818,-73.040,-176.674,8.148,148.622
C00660=1170.707,315.066,-73.072,-176.672,8.151,148.622
C00661=1170.703,315.314,-73.103,-176.669,8.154,148.622
C00662=1170.699,315.562,-73.134,-176.667,8.158,148.622
C00663=1170.695,315.810,-73.165,-176.664,8.161,148.622
C00664=1170.691,316.058,-73.197,-176.662,8.164,148.622
C00665=1170.687,316.306,-73.228,-176.659,8.167,148.622
C00666=1170.682,316.554,-73.260,-176.657,8.170,148.623
C00667=1170.678,316.802,-73.291,-176.654,8.173,148.623
C00668=1170.675,317.050,-73.323,-176.651,8.177,148.623
C00669=1170.670,317.298,-73.354,-176.649,8.181,148.623
C00670=1170.666,317.546,-73.385,-176.646,8.184,148.623
C00671=1170.662,317.794,-73.417,-176.644,8.187,148.623
C00672=1170.658,318.042,-73.449,-176.641,8.190,148.623
C00673=1170.653,318.290,-73.480,-176.639,8.193,148.623
C00674=1170.649,318.538,-73.512,-176.636,8.196,148.623
C00675=1170.645,318.785,-73.543,-176.634,8.200,148.624
C00676=1170.641,319.034,-73.574,-176.631,8.203,148.624
C00677=1170.637,319.282,-73.606,-176.629,8.206,148.624
C00678=1170.633,319.529,-73.638,-176.626,8.209,148.624
C00679=1170.628,319.778,-73.670,-176.624,8.212,148.624
C00680=1170.624,320.026,-73.701,-176.621,8.215,148.624
C00681=1170.620,320.274,-73.733,-176.619,8.218,148.624
C00682=1170.616,320.522,-73.764,-176.616,8.222,148.624
C00683=1170.612,320.769,-73.796,-176.614,8.225,148.624
C00684=1170.608,321.017,-73.828,-176.611,8.229,148.625
C00685=1170.603,321.265,-73.859,-176.608,8.232,148.625
C00686=1170.599,321.513,-73.891,-176.606,8.235,148.625
C00687=1170.596,321.761,-73.923,-176.603,8.238,148.625
C00688=1170.591,322.009,-73.955,-176.601,8.241,148.625
C00689=1170.587,322.257,-73.987,-176.599,8.245,148.625
C00690=1170.583,322.505,-74.019,-176.596,8.248,148.625
C00691=1170.579,322.752,-74.050,-176.594,8.251,148.625
C00692=1170.574,323.001,-74.083,-176.591,8.254,148.625
C00693=1170.571,323.249,-74.114,-176.589,8.257,148.626
C00694=1170.566,323.496,-74.146,-176.586,8.261,148.626
C00695=1170.562,323.745,-74.178,-176.584,8.264,148.626
C00696=1170.558,323.993,-74.209,-176.581,8.268,148.626
C00697=1170.554,324.241,-74.241,-176.578,8.271,148.626
C00698=1170.550,324.489,-74.273,-176.576,8.274,148.626
C00699=1170.546,324.736,-74.306,-176.573,8.277,148.626
C00700=1170.541,324.984,-74.337,-176.571,8.280,148.626
C00701=1170.537,325.232,-74.370,-176.568,8.283,148.627
C00702=1170.533,325.480,-74.402,-176.566,8.286,148.627
C00703=1170.530,325.728,-74.434,-176.563,8.290,148.627
C00704=1170.525,325.976,-74.466,-176.561,8.293,148.627
C00705=1170.521,326.224,-74.497,-176.558,8.296,148.627
C00706=1170.516,326.472,-74.530,-176.555,8.300,148.627
C00707=1170.512,326.719,-74.561,-176.553,8.303,148.627
C00708=1170.508,326.967,-74.593,-176.550,8.306,148.627
C00709=1170.504,327.215,-74.626,-176.548,8.310,148.628
C00710=1170.501,327.463,-74.658,-176.546,8.313,148.628
C00711=1170.496,327.711,-74.690,-176.543,8.316,148.628
C00712=1170.492,327.959,-74.722,-176.541,8.319,148.628
C00713=1170.487,328.207,-74.755,-176.539,8.323,148.628
C00714=1170.484,328.455,-74.787,-176.536,8.326,148.628
C00715=1170.479,328.702,-74.819,-176.533,8.330,148.628
C00716=1170.475,328.950,-74.851,-176.531,8.333,148.629
C00717=1170.471,329.199,-74.883,-176.528,8.336,148.629
C00718=1170.467,329.446,-74.916,-176.526,8.339,148.629
C00719=1170.463,329.695,-74.948,-176.523,8.343,148.629
C00720=1170.459,329.942,-74.980,-176.521,8.346,148.629
C00721=1170.454,330.190,-75.012,-176.518,8.349,148.629
C00722=1170.451,330.438,-75.045,-176.516,8.352,148.629
C00723=1170.446,330.686,-75.077,-176.513,8.356,148.630
C00724=1170.443,330.933,-75.110,-176.511,8.359,148.630
C00725=1170.438,331.181,-75.142,-176.508,8.363,148.630
C00726=1170.433,331.429,-75.174,-176.506,8.366,148.630
C00727=1170.430,331.677,-75.207,-176.503,8.369,148.630
C00728=1170.426,331.925,-75.239,-176.501,8.372,148.630
C00729=1170.422,332.173,-75.272,-176.499,8.375,148.631
C00730=1170.418,332.421,-75.304,-176.496,8.379,148.631
C00731=1170.413,332.669,-75.337,-176.493,8.383,148.631
C00732=1170.409,332.916,-75.369,-176.491,8.386,148.631
C00733=1170.405,333.164,-75.402,-176.489,8.389,148.631
C00734=1170.401,333.412,-75.435,-176.486,8.393,148.631
C00735=1170.397,333.660,-75.467,-176.484,8.395,148.631
C00736=1170.393,333.908,-75.500,-176.481,8.399,148.632
C00737=1170.389,334.156,-75.533,-176.479,8.402,148.632
C00738=1170.385,334.404,-75.565,-176.476,8.406,148.632
C00739=1170.381,334.651,-75.598,-176.474,8.410,148.632
C00740=1170.376,334.899,-75.630,-176.471,8.412,148.632
C00741=1170.372,335.146,-75.663,-176.469,8.416,148.632
C00742=1170.368,335.395,-75.695,-176.467,8.419,148.633
C00743=1170.364,335.642,-75.728,-176.464,8.422,148.633
C00744=1170.360,335.890,-75.761,-176.462,8.426,148.633
C00745=1170.356,336.138,-75.793,-176.459,8.429,148.633
C00746=1170.352,336.386,-75.826,-176.456,8.433,148.633
C00747=1170.348,336.634,-75.859,-176.454,8.436,148.634
C00748=1170.343,336.882,-75.892,-176.452,8.439,148.634
C00749=1170.340,337.129,-75.924,-176.450,8.443,148.634
C00750=1170.336,337.377,-75.958,-176.447,8.446,148.634
C00751=1170.332,337.625,-75.991,-176.444,8.450,148.634
C00752=1170.327,337.873,-76.023,-176.442,8.453,148.634
C00753=1170.323,338.121,-76.056,-176.439,8.456,148.635
C00754=1170.320,338.368,-76.089,-176.437,8.460,148.635
C00755=1170.316,338.616,-76.122,-176.435,8.463,148.635
C00756=1170.311,338.865,-76.154,-176.433,8.466,148.635
C00757=1170.307,339.112,-76.188,-176.429,8.470,148.635
C00758=1170.303,339.360,-76.221,-176.427,8.473,148.636
C00759=1170.298,339.639,-76.258,-176.424,8.478,148.636
C00760=1170.294,339.918,-76.295,-176.422,8.481,148.636
C00761=1170.289,340.198,-76.332,-176.419,8.485,148.636
C00762=1170.284,340.477,-76.370,-176.416,8.489,148.637
C00763=1170.279,340.725,-76.402,-176.414,8.492,148.637
C00764=1170.275,340.973,-76.435,-176.412,8.496,148.637
C00765=1170.271,341.220,-76.468,-176.409,8.499,148.637
C00766=1170.268,341.469,-76.502,-176.407,8.502,148.637
C00767=1170.264,341.717,-76.535,-176.404,8.506,148.637
C00768=1170.259,341.964,-76.568,-176.401,8.509,148.638
C00769=1170.255,342.212,-76.601,-176.399,8.513,148.638
C00770=1170.251,342.460,-76.634,-176.397,8.516,148.638
C00771=1170.247,342.707,-76.668,-176.395,8.519,148.638
C00772=1170.243,342.955,-76.701,-176.392,8.523,148.639
C00773=1170.239,343.203,-76.734,-176.389,8.527,148.639
C00774=1170.235,343.451,-76.767,-176.387,8.530,148.639
C00775=1170.230,343.698,-76.800,-176.385,8.533,148.639
C00776=1170.226,343.946,-76.833,-176.383,8.537,148.639
C00777=1170.222,344.193,-76.867,-176.380,8.541,148.640
C00778=1170.218,344.441,-76.900,-176.377,8.544,148.640
C00779=1170.214,344.689,-76.934,-176.375,8.547,148.640
C00780=1170.210,344.936,-76.967,-176.373,8.551,148.640
C00781=1170.207,345.185,-77.000,-176.371,8.554,148.640
C00782=1170.202,345.433,-77.033,-176.368,8.558,148.641
C00783=1170.198,345.680,-77.067,-176.365,8.561,148.641
C00784=1170.194,345.927,-77.100,-176.363,8.565,148.641
C00785=1170.190,346.175,-77.134,-176.361,8.568,148.641
C00786=1170.186,346.423,-77.167,-176.358,8.572,148.642
C00787=1170.182,346.671,-77.200,-176.356,8.575,148.642
C00788=1170.177,346.919,-77.234,-176.353,8.579,148.642
C00789=1170.174,347.166,-77.268,-176.351,8.582,148.642
C00790=1170.170,347.414,-77.301,-176.349,8.585,148.643
C00791=1170.166,347.662,-77.334,-176.346,8.589,148.643
C00792=1170.162,347.909,-77.368,-176.344,8.593,148.643
C00793=1170.158,348.157,-77.401,-176.341,8.596,148.643
C00794=1170.153,348.405,-77.435,-176.339,8.599,148.643
C00795=1170.150,348.653,-77.469,-176.336,8.603,148.644
C00796=1170.145,348.900,-77.502,-176.334,8.607,148.644
C00797=1170.141,349.148,-77.536,-176.332,8.610,148.644
C00798=1170.137,349.395,-77.569,-176.330,8.614,148.645
C00799=1170.133,349.643,-77.603,-176.327,8.618,148.645
C00800=1170.129,349.892,-77.637,-176.325,8.621,148.645
C00801=1170.125,350.139,-77.671,-176.322,8.624,148.645
C00802=1170.121,350.386,-77.704,-176.320,8.628,148.645
C00803=1170.116,350.634,-77.738,-176.317,8.632,148.646
C00804=1170.113,350.882,-77.772,-176.315,8.635,148.646
C00805=1170.109,351.129,-77.806,-176.313,8.638,148.646
C00806=1170.105,351.377,-77.839,-176.311,8.642,148.647
C00807=1170.100,351.625,-77.873,-176.308,8.646,148.647
C00808=1170.096,351.872,-77.906,-176.306,8.649,148.647
C00809=1170.093,352.120,-77.941,-176.303,8.653,148.647
C00810=1170.089,352.368,-77.974,-176.301,8.656,148.647
C00811=1170.084,352.615,-78.008,-176.298,8.660,148.648
C00812=1170.081,352.864,-78.042,-176.296,8.664,148.648
C00813=1170.077,353.111,-78.076,-176.294,8.667,148.648
C00814=1170.072,353.358,-78.110,-176.292,8.670,148.649
C00815=1170.068,353.606,-78.143,-176.289,8.674,148.649
C00816=1170.064,353.854,-78.178,-176.287,8.678,148.649
C00817=1170.060,354.101,-78.212,-176.285,8.681,148.649
C00818=1170.056,354.349,-78.245,-176.282,8.685,148.650
C00819=1170.052,354.597,-78.280,-176.280,8.689,148.650
C00820=1170.049,354.844,-78.314,-176.277,8.692,148.650
C00821=1170.044,355.092,-78.347,-176.276,8.696,148.651
C00822=1170.040,355.340,-78.382,-176.273,8.700,148.651
C00823=1170.037,355.587,-78.416,-176.270,8.703,148.651
C00824=1170.032,355.835,-78.449,-176.268,8.706,148.651
C00825=1170.028,356.083,-78.484,-176.266,8.711,148.652
C00826=1170.024,356.330,-78.518,-176.264,8.714,148.652
C00827=1170.020,356.577,-78.552,-176.261,8.717,148.652
C00828=1170.017,356.825,-78.586,-176.259,8.721,148.653
C00829=1170.012,357.073,-78.620,-176.257,8.725,148.653
C00830=1170.008,357.320,-78.654,-176.254,8.728,148.653
C00831=1170.004,357.569,-78.689,-176.252,8.732,148.654
C00832=1170.000,357.816,-78.723,-176.250,8.736,148.654
C00833=1169.996,358.064,-78.757,-176.247,8.739,148.654
C00834=1169.993,358.311,-78.791,-176.245,8.743,148.654
C00835=1169.988,358.558,-78.826,-176.243,8.747,148.655
C00836=1169.984,358.807,-78.859,-176.240,8.750,148.655
C00837=1169.980,359.054,-78.894,-176.238,8.754,148.655
C00838=1169.977,359.302,-78.928,-176.236,8.757,148.656
C00839=1169.972,359.549,-78.962,-176.233,8.762,148.656
C00840=1169.967,359.797,-78.997,-176.231,8.765,148.656
C00841=1169.964,360.045,-79.031,-176.229,8.768,148.657
C00842=1169.960,360.292,-79.066,-176.227,8.773,148.657
C00843=1169.956,360.540,-79.100,-176.224,8.776,148.657
C00844=1169.952,360.787,-79.134,-176.223,8.780,148.658
C00845=1169.949,361.035,-79.169,-176.220,8.784,148.658
C00846=1169.944,361.282,-79.203,-176.218,8.787,148.658
C00847=1169.940,361.531,-79.238,-176.216,8.791,148.659
C00848=1169.936,361.778,-79.272,-176.213,8.795,148.659
C00849=1169.932,362.025,-79.306,-176.211,8.799,148.659
C00850=1169.928,362.273,-79.342,-176.209,8.802,148.660
C00851=1169.924,362.520,-79.376,-176.207,8.805,148.660
C00852=1169.920,362.768,-79.410,-176.204,8.810,148.660
C00853=1169.916,363.015,-79.445,-176.202,8.813,148.661
C00854=1169.912,363.263,-79.479,-176.200,8.817,148.661
C00855=1169.908,363.511,-79.514,-176.198,8.821,148.662
C00856=1169.904,363.759,-79.548,-176.196,8.825,148.662
C00857=1169.900,364.005,-79.583,-176.194,8.828,148.662
C00858=1169.896,364.253,-79.618,-176.192,8.832,148.663
C00859=1169.892,364.501,-79.653,-176.189,8.836,148.663
C00860=1169.889,364.748,-79.687,-176.187,8.839,148.663
C00861=1169.885,364.996,-79.722,-176.185,8.843,148.664
C00862=1169.880,365.243,-79.757,-176.183,8.847,148.664
C00863=1169.876,365.526,-79.796,-176.181,8.851,148.665
C00864=1169.871,365.807,-79.836,-176.179,8.855,148.665
C00865=1169.867,366.090,-79.876,-176.176,8.860,148.666
C00866=1169.862,366.373,-79.915,-176.174,8.864,148.666
C00867=1169.858,366.620,-79.950,-176.172,8.868,148.667
C00868=1169.855,366.867,-79.984,-176.170,8.872,148.667
C00869=1169.850,367.115,-80.019,-176.168,8.875,148.667
C00870=1169.847,367.362,-80.054,-176.166,8.878,148.668
C00871=1169.842,367.610,-80.089,-176.163,8.883,148.668
C00872=1169.838,367.857,-80.124,-176.162,8.887,148.668
C00873=1169.835,368.105,-80.158,-176.160,8.890,148.669
C00874=1169.831,368.352,-80.193,-176.158,8.894,148.670
C00875=1169.827,368.600,-80.228,-176.157,8.898,148.670
C00876=1169.822,368.847,-80.263,-176.155,8.901,148.670
C00877=1169.819,369.095,-80.298,-176.153,8.905,148.671
C00878=1169.815,369.343,-80.333,-176.150,8.909,148.671
C00879=1169.810,369.590,-80.368,-176.149,8.913,148.672
C00880=1169.806,369.838,-80.403,-176.147,8.916,148.672
C00881=1169.803,370.084,-80.438,-176.145,8.920,148.673
C00882=1169.799,370.332,-80.473,-176.143,8.924,148.673
C00883=1169.795,370.580,-80.508,-176.142,8.928,148.674
C00884=1169.791,370.827,-80.543,-176.140,8.931,148.674
C00885=1169.787,371.075,-80.578,-176.138,8.935,148.675
C00886=1169.783,371.322,-80.614,-176.136,8.939,148.675
C00887=1169.779,371.570,-80.648,-176.135,8.942,148.676
C00888=1169.775,371.817,-80.684,-176.133,8.946,148.676
C00889=1169.771,372.065,-80.719,-176.131,8.950,148.677
C00890=1169.767,372.312,-80.754,-176.130,8.954,148.677
C00891=1169.763,372.560,-80.789,-176.128,8.957,148.678
C00892=1169.759,372.808,-80.824,-176.127,8.961,148.678
C00893=1169.755,373.055,-80.859,-176.125,8.965,148.679
C00894=1169.751,373.302,-80.895,-176.123,8.969,148.679
C00895=1169.747,373.550,-80.930,-176.122,8.972,148.680
C00896=1169.743,373.797,-80.965,-176.120,8.976,148.680
C00897=1169.740,374.045,-81.001,-176.119,8.979,148.681
C00898=1169.736,374.293,-81.035,-176.117,8.983,148.681
C00899=1169.731,374.539,-81.071,-176.116,8.987,148.682
C00900=1169.728,374.787,-81.106,-176.115,8.991,148.683
C00901=1169.724,375.034,-81.142,-176.113,8.994,148.683
C00902=1169.720,375.283,-81.176,-176.111,8.998,148.684
C00903=1169.716,375.529,-81.212,-176.110,9.001,148.684
C00904=1169.712,375.777,-81.247,-176.109,9.005,148.685
C00905=1169.708,376.024,-81.283,-176.107,9.009,148.685
C00906=1169.704,376.272,-81.317,-176.106,9.013,148.686
C00907=1169.700,376.519,-81.353,-176.105,9.016,148.687
C00908=1169.696,376.767,-81.389,-176.104,9.020,148.687
C00909=1169.692,377.015,-81.424,-176.102,9.024,148.688
C00910=1169.688,377.261,-81.460,-176.101,9.027,148.688
C00911=1169.684,377.509,-81.495,-176.100,9.031,148.689
C00912=1169.681,377.756,-81.531,-176.098,9.035,148.690
C00913=1169.677,378.005,-81.566,-176.098,9.038,148.690
C00914=1169.672,378.251,-81.601,-176.096,9.042,148.691
C00915=1169.669,378.499,-81.636,-176.095,9.045,148.691
C00916=1169.664,378.747,-81.672,-176.094,9.049,148.692
C00917=1169.661,378.994,-81.708,-176.092,9.053,148.693
C00918=1169.657,379.242,-81.744,-176.092,9.056,148.693
C00919=1169.653,379.488,-81.779,-176.091,9.060,148.694
C00920=1169.649,379.736,-81.814,-176.090,9.063,148.695
C00921=1169.645,379.983,-81.850,-176.088,9.067,148.695
C00922=1169.641,380.231,-81.886,-176.088,9.070,148.696
C00923=1169.637,380.478,-81.921,-176.087,9.073,148.697
C00924=1169.633,380.726,-81.957,-176.086,9.077,148.697
C00925=1169.629,380.973,-81.992,-176.085,9.080,148.698
C00926=1169.626,381.221,-82.028,-176.084,9.085,148.699
C00927=1169.621,381.468,-82.064,-176.083,9.088,148.699
C00928=1169.617,381.715,-82.099,-176.083,9.091,148.700
C00929=1169.613,381.963,-82.135,-176.082,9.094,148.701
C00930=1169.610,382.210,-82.170,-176.080,9.098,148.701
C00931=1169.606,382.458,-82.206,-176.080,9.101,148.702
C00932=1169.602,382.705,-82.242,-176.079,9.105,148.703
C00933=1169.598,382.953,-82.277,-176.079,9.108,148.703
C00934=1169.594,383.200,-82.313,-176.077,9.112,148.704
C00935=1169.590,383.447,-82.348,-176.077,9.115,148.705
C00936=1169.586,383.695,-82.384,-176.076,9.119,148.706
C00937=1169.582,383.943,-82.420,-176.076,9.122,148.706
C00938=1169.578,384.190,-82.455,-176.075,9.125,148.707
C00939=1169.575,384.438,-82.491,-176.074,9.128,148.707
C00940=1169.570,384.684,-82.527,-176.074,9.132,148.708
C00941=1169.566,384.932,-82.563,-176.073,9.135,148.709
C00942=1169.563,385.179,-82.599,-176.073,9.138,148.710
C00943=1169.558,385.427,-82.635,-176.072,9.141,148.710
C00944=1169.555,385.674,-82.670,-176.072,9.145,148.711
C00945=1169.551,385.922,-82.706,-176.071,9.148,148.712
C00946=1169.547,386.169,-82.743,-176.071,9.152,148.713
C00947=1169.543,386.416,-82.778,-176.070,9.155,148.713
C00948=1169.539,386.663,-82.813,-176.070,9.157,148.714
C00949=1169.535,386.911,-82.849,-176.070,9.161,148.715
C00950=1169.531,387.159,-82.885,-176.069,9.164,148.716
C00951=1169.527,387.406,-82.921,-176.069,9.167,148.716
C00952=1169.524,387.653,-82.957,-176.069,9.170,148.717
C00953=1169.519,387.901,-82.993,-176.068,9.173,148.718
C00954=1169.516,388.148,-83.029,-176.068,9.176,148.718
C00955=1169.511,388.395,-83.064,-176.068,9.179,148.719
C00956=1169.507,388.642,-83.101,-176.068,9.182,148.720
C00957=1169.504,388.890,-83.136,-176.068,9.185,148.721
C00958=1169.500,389.137,-83.172,-176.067,9.188,148.721
C00959=1169.496,389.385,-83.208,-176.067,9.192,148.722
C00960=1169.492,389.632,-83.244,-176.067,9.194,148.723
C00961=1169.489,389.880,-83.280,-176.067,9.197,148.724
C00962=1169.484,390.127,-83.316,-176.067,9.200,148.724
C00963=1169.481,390.375,-83.351,-176.067,9.203,148.725
C00964=1169.476,390.622,-83.388,-176.067,9.206,148.726
C00965=1169.472,390.869,-83.423,-176.067,9.209,148.726
C00966=1169.469,391.116,-83.459,-176.067,9.211,148.727
C00967=1169.465,391.401,-83.501,-176.067,9.215,148.728
C00968=1169.460,391.687,-83.542,-176.066,9.218,148.729
C00969=1169.455,391.971,-83.584,-176.067,9.221,148.730
C00970=1169.451,392.257,-83.625,-176.067,9.225,148.731
C00971=1169.447,392.503,-83.660,-176.067,9.227,148.731
C00972=1169.443,392.751,-83.697,-176.067,9.230,148.732
C00973=1169.439,392.998,-83.733,-176.067,9.234,148.733
C00974=1169.434,393.246,-83.769,-176.067,9.236,148.734
C00975=1169.431,393.493,-83.805,-176.067,9.239,148.734
C00976=1169.427,393.740,-83.841,-176.067,9.241,148.735
C00977=1169.423,393.988,-83.877,-176.068,9.244,148.736
C00978=1169.420,394.235,-83.913,-176.068,9.246,148.737
C00979=1169.415,394.483,-83.949,-176.068,9.249,148.737
C00980=1169.412,394.730,-83.986,-176.068,9.252,148.738
C00981=1169.408,394.978,-84.022,-176.068,9.254,148.739
C00982=1169.404,395.225,-84.057,-176.068,9.257,148.739
C00983=1169.401,395.472,-84.094,-176.068,9.259,148.740
C00984=1169.396,395.720,-84.130,-176.069,9.262,148.741
C00985=1169.392,395.967,-84.165,-176.069,9.264,148.742
C00986=1169.388,396.214,-84.202,-176.069,9.267,148.742
C00987=1169.384,396.461,-84.237,-176.069,9.270,148.743
C00988=1169.380,396.708,-84.274,-176.070,9.272,148.744
C00989=1169.376,396.956,-84.310,-176.070,9.275,148.745
C00990=1169.372,397.204,-84.346,-176.070,9.278,148.745
C00991=1169.369,397.451,-84.382,-176.071,9.279,148.746
C00992=1169.365,397.698,-84.418,-176.071,9.282,148.747
C00993=1169.361,397.945,-84.454,-176.071,9.284,148.747
C00994=1169.357,398.193,-84.490,-176.071,9.287,148.748
C00995=1169.353,398.441,-84.526,-176.071,9.290,148.749
C00996=1169.349,398.687,-84.562,-176.072,9.291,148.750
C00997=1169.345,398.935,-84.599,-176.072,9.294,148.750
C00998=1169.342,399.182,-84.635,-176.072,9.296,148.751
C00999=1169.337,399.430,-84.671,-176.072,9.299,148.752
C01000=1169.334,399.677,-84.707,-176.073,9.301,148.752
C01001=1169.329,399.925,-84.743,-176.073,9.303,148.753
C01002=1169.326,400.172,-84.780,-176.073,9.306,148.754
C01003=1169.322,400.419,-84.816,-176.074,9.308,148.754
C01004=1169.318,400.667,-84.851,-176.074,9.310,148.755
C01005=1169.314,400.914,-84.888,-176.074,9.313,148.756
C01006=1169.310,401.161,-84.923,-176.075,9.315,148.756
C01007=1169.306,401.408,-84.960,-176.075,9.317,148.757
C01008=1169.302,401.656,-84.996,-176.076,9.319,148.758
C01009=1169.298,401.903,-85.033,-176.076,9.321,148.759
C01010=1169.294,402.150,-85.068,-176.076,9.324,148.759
C01011=1169.290,402.397,-85.105,-176.076,9.325,148.760
C01012=1169.286,402.645,-85.141,-176.077,9.328,148.760
C01013=1169.282,402.892,-85.177,-176.077,9.330,148.761
C01014=1169.279,403.140,-85.213,-176.077,9.332,148.762
C01015=1169.275,403.387,-85.250,-176.078,9.334,148.762
C01016=1169.271,403.634,-85.285,-176.078,9.337,148.763
C01017=1169.267,403.881,-85.322,-176.079,9.338,148.764
C01018=1169.263,404.129,-85.358,-176.079,9.341,148.764
C01019=1169.259,404.376,-85.395,-176.080,9.342,148.765
C01020=1169.255,404.624,-85.430,-176.080,9.345,148.766
C01021=1169.251,404.871,-85.467,-176.080,9.347,148.766
C01022=1169.248,405.118,-85.503,-176.080,9.349,148.767
C01023=1169.244,405.366,-85.539,-176.081,9.351,148.768
C01024=1169.240,405.613,-85.575,-176.081,9.353,148.768
C01025=1169.236,405.860,-85.612,-176.082,9.355,148.769
C01026=1169.232,406.108,-85.647,-176.082,9.357,148.770
C01027=1169.228,406.355,-85.684,-176.082,9.359,148.770
C01028=1169.224,406.602,-85.720,-176.083,9.361,148.771
C01029=1169.220,406.850,-85.757,-176.083,9.363,148.771
C01030=1169.217,407.097,-85.792,-176.084,9.365,148.772
C01031=1169.213,407.344,-85.829,-176.084,9.367,148.773
C01032=1169.209,407.592,-85.865,-176.084,9.369,148.773
C01033=1169.205,407.839,-85.902,-176.085,9.371,148.774
C01034=1169.201,408.087,-85.937,-176.085,9.373,148.775
C01035=1169.197,408.334,-85.974,-176.085,9.375,148.775
C01036=1169.193,408.581,-86.009,-176.086,9.377,148.776
C01037=1169.189,408.828,-86.046,-176.086,9.379,148.776
C01038=1169.186,409.076,-86.082,-176.086,9.381,148.777
C01039=1169.181,409.323,-86.119,-176.087,9.382,148.777
C01040=1169.177,409.570,-86.156,-176.087,9.385,148.778
C01041=1169.174,409.818,-86.191,-176.087,9.386,148.779
C01042=1169.170,410.065,-86.228,-176.088,9.388,148.779
C01043=1169.166,410.312,-86.264,-176.089,9.390,148.780
C01044=1169.162,410.560,-86.300,-176.089,9.392,148.780
C01045=1169.158,410.807,-86.336,-176.089,9.394,148.781
C01046=1169.154,411.054,-86.373,-176.090,9.395,148.782
C01047=1169.150,411.302,-86.408,-176.090,9.398,148.782
C01048=1169.146,411.549,-86.445,-176.090,9.399,148.783
C01049=1169.143,411.796,-86.481,-176.091,9.401,148.783
C01050=1169.139,412.044,-86.518,-176.091,9.404,148.784
C01051=1169.135,412.291,-86.554,-176.091,9.405,148.785
C01052=1169.131,412.538,-86.590,-176.092,9.407,148.785
C01053=1169.127,412.786,-86.627,-176.092,9.408,148.786
C01054=1169.123,413.033,-86.662,-176.092,9.411,148.786
C01055=1169.119,413.280,-86.699,-176.093,9.412,148.787
C01056=1169.116,413.527,-86.736,-176.093,9.414,148.787
C01057=1169.111,413.775,-86.772,-176.093,9.416,148.788
C01058=1169.107,414.022,-86.809,-176.093,9.418,148.788
C01059=1169.103,414.270,-86.844,-176.094,9.419,148.789
C01060=1169.099,414.517,-86.881,-176.094,9.421,148.790
C01061=1169.096,414.764,-86.917,-176.094,9.423,148.790
C01062=1169.092,415.012,-86.953,-176.095,9.425,148.791
C01063=1169.088,415.258,-86.990,-176.095,9.427,148.791
C01064=1169.084,415.506,-87.026,-176.096,9.428,148.792
C01065=1169.082,415.754,-87.062,-176.095,9.430,148.792
C01066=1169.080,416.001,-87.098,-176.096,9.432,148.793
C01067=1169.079,416.295,-87.141,-176.096,9.433,148.793
C01068=1169.081,416.590,-87.183,-176.096,9.436,148.794
C01069=1169.083,416.883,-87.226,-176.097,9.437,148.795
C01070=1169.087,417.177,-87.269,-176.097,9.439,148.795
C01071=1168.665,417.179,-87.314,-176.101,9.450,148.799
C01072=1168.662,416.882,-87.271,-176.100,9.448,148.798
C01073=1168.660,416.585,-87.228,-176.100,9.447,148.798
C01074=1168.659,416.287,-87.184,-176.100,9.444,148.797
C01075=1168.660,415.989,-87.141,-176.099,9.443,148.797
C01076=1168.662,415.742,-87.105,-176.099,9.441,148.796
C01077=1168.664,415.495,-87.069,-176.099,9.439,148.796
C01078=1168.667,415.248,-87.033,-176.098,9.437,148.795
C01079=1168.671,415.000,-86.997,-176.098,9.436,148.794
C01080=1168.675,414.753,-86.960,-176.097,9.434,148.794
C01081=1168.679,414.506,-86.924,-176.098,9.432,148.793
C01082=1168.683,414.258,-86.888,-176.097,9.430,148.793
C01083=1168.686,414.011,-86.851,-176.097,9.429,148.792
C01084=1168.690,413.763,-86.814,-176.096,9.427,148.792
C01085=1168.694,413.516,-86.779,-176.096,9.425,148.791
C01086=1168.698,413.269,-86.742,-176.095,9.423,148.790
C01087=1168.702,413.021,-86.706,-176.095,9.421,148.790
C01088=1168.706,412.774,-86.669,-176.094,9.420,148.789
C01089=1168.710,412.526,-86.633,-176.095,9.417,148.789
C01090=1168.713,412.279,-86.597,-176.094,9.416,148.788
C01091=1168.717,412.032,-86.560,-176.094,9.414,148.788
C01092=1168.721,411.785,-86.525,-176.094,9.412,148.787
C01093=1168.725,411.538,-86.488,-176.093,9.410,148.787
C01094=1168.729,411.290,-86.452,-176.093,9.408,148.786
C01095=1168.733,411.043,-86.415,-176.092,9.407,148.785
C01096=1168.737,410.796,-86.378,-176.092,9.404,148.785
C01097=1168.741,410.548,-86.343,-176.091,9.403,148.784
C01098=1168.745,410.301,-86.306,-176.091,9.401,148.784
C01099=1168.748,410.053,-86.270,-176.091,9.399,148.783
C01100=1168.752,409.806,-86.234,-176.091,9.397,148.782
C01101=1168.756,409.559,-86.198,-176.090,9.396,148.782
C01102=1168.760,409.312,-86.161,-176.090,9.393,148.781
C01103=1168.764,409.064,-86.126,-176.090,9.392,148.781
C01104=1168.768,408.817,-86.089,-176.089,9.390,148.780
C01105=1168.772,408.570,-86.052,-176.089,9.387,148.779
C01106=1168.776,408.322,-86.016,-176.088,9.386,148.779
C01107=1168.780,408.075,-85.980,-176.088,9.384,148.778
C01108=1168.784,407.828,-85.944,-176.088,9.381,148.777
C01109=1168.788,407.580,-85.907,-176.087,9.380,148.777
C01110=1168.791,407.333,-85.872,-176.087,9.378,148.776
C01111=1168.795,407.086,-85.835,-176.086,9.376,148.776
C01112=1168.799,406.838,-85.799,-176.086,9.374,148.775
C01113=1168.803,406.591,-85.762,-176.085,9.373,148.775
C01114=1168.807,406.343,-85.727,-176.085,9.370,148.774
C01115=1168.811,406.096,-85.690,-176.085,9.368,148.773
C01116=1168.815,405.849,-85.654,-176.085,9.366,148.772
C01117=1168.819,405.602,-85.617,-176.084,9.364,148.772
C01118=1168.822,405.355,-85.581,-176.084,9.362,148.771
C01119=1168.826,405.107,-85.545,-176.083,9.360,148.771
C01120=1168.830,404.860,-85.509,-176.083,9.358,148.770
C01121=1168.834,404.612,-85.473,-176.083,9.356,148.769
C01122=1168.838,404.365,-85.436,-176.082,9.354,148.769
C01123=1168.842,404.117,-85.400,-176.082,9.351,148.768
C01124=1168.845,403.871,-85.364,-176.081,9.350,148.767
C01125=1168.850,403.624,-85.328,-176.081,9.347,148.767
C01126=1168.854,403.377,-85.292,-176.081,9.346,148.766
C01127=1168.858,403.129,-85.256,-176.080,9.343,148.765
C01128=1168.862,402.882,-85.219,-176.080,9.341,148.765
C01129=1168.866,402.634,-85.183,-176.080,9.339,148.764
C01130=1168.870,402.387,-85.147,-176.079,9.337,148.763
C01131=1168.874,402.139,-85.111,-176.079,9.334,148.763
C01132=1168.878,401.892,-85.074,-176.078,9.333,148.762
C01133=1168.881,401.645,-85.039,-176.078,9.330,148.761
C01134=1168.886,401.397,-85.002,-176.078,9.327,148.761
C01135=1168.889,401.150,-84.966,-176.077,9.326,148.760
C01136=1168.893,400.903,-84.931,-176.077,9.323,148.759
C01137=1168.897,400.655,-84.894,-176.076,9.322,148.759
C01138=1168.900,400.408,-84.858,-176.076,9.319,148.758
C01139=1168.905,400.161,-84.821,-176.076,9.317,148.757
C01140=1168.908,399.913,-84.786,-176.075,9.315,148.757
C01141=1168.912,399.666,-84.749,-176.075,9.312,148.756
C01142=1168.916,399.418,-84.713,-176.075,9.310,148.755
C01143=1168.920,399.171,-84.677,-176.074,9.308,148.754
C01144=1168.924,398.924,-84.641,-176.074,9.305,148.754
C01145=1168.928,398.677,-84.604,-176.074,9.302,148.753
C01146=1168.932,398.429,-84.569,-176.074,9.300,148.752
C01147=1168.936,398.181,-84.532,-176.073,9.298,148.752
C01148=1168.939,397.934,-84.496,-176.073,9.296,148.751
C01149=1168.944,397.687,-84.460,-176.073,9.293,148.750
C01150=1168.947,397.440,-84.424,-176.072,9.290,148.749
C01151=1168.951,397.192,-84.388,-176.072,9.288,148.749
C01152=1168.955,396.945,-84.351,-176.072,9.286,148.748
C01153=1168.959,396.697,-84.315,-176.071,9.284,148.747
C01154=1168.963,396.450,-84.280,-176.071,9.281,148.747
C01155=1168.967,396.204,-84.244,-176.071,9.278,148.746
C01156=1168.971,395.956,-84.208,-176.071,9.276,148.745
C01157=1168.975,395.709,-84.171,-176.071,9.273,148.745
C01158=1168.979,395.461,-84.135,-176.071,9.271,148.744
C01159=1168.983,395.214,-84.100,-176.070,9.268,148.743
C01160=1168.987,394.966,-84.063,-176.070,9.265,148.742
C01161=1168.990,394.719,-84.027,-176.070,9.263,148.741
C01162=1168.995,394.471,-83.991,-176.070,9.260,148.741
C01163=1168.998,394.224,-83.955,-176.070,9.258,148.740
C01164=1169.002,393.977,-83.919,-176.069,9.255,148.739
C01165=1169.006,393.729,-83.882,-176.069,9.252,148.739
C01166=1169.010,393.482,-83.847,-176.069,9.250,148.738
C01167=1169.014,393.234,-83.811,-176.069,9.247,148.737
C01168=1169.017,392.987,-83.775,-176.069,9.245,148.736
C01169=1169.022,392.739,-83.738,-176.069,9.241,148.736
C01170=1169.026,392.493,-83.703,-176.069,9.239,148.735
C01171=1169.029,392.246,-83.667,-176.068,9.236,148.734
C01172=1169.034,391.960,-83.626,-176.069,9.233,148.733
C01173=1169.038,391.676,-83.584,-176.068,9.230,148.732
C01174=1169.043,391.391,-83.543,-176.069,9.226,148.732
C01175=1169.047,391.105,-83.501,-176.068,9.223,148.731
C01176=1169.051,390.858,-83.465,-176.069,9.220,148.730
C01177=1169.055,390.610,-83.429,-176.068,9.217,148.729
C01178=1169.059,390.363,-83.394,-176.069,9.214,148.728
C01179=1169.063,390.116,-83.357,-176.069,9.211,148.728
C01180=1169.067,389.869,-83.321,-176.069,9.209,148.727
C01181=1169.071,389.621,-83.286,-176.069,9.206,148.726
C01182=1169.075,389.374,-83.249,-176.069,9.203,148.726
C01183=1169.078,389.126,-83.213,-176.069,9.200,148.725
C01184=1169.082,388.879,-83.178,-176.069,9.197,148.724
C01185=1169.087,388.631,-83.142,-176.070,9.194,148.723
C01186=1169.090,388.384,-83.105,-176.070,9.190,148.723
C01187=1169.094,388.136,-83.069,-176.070,9.188,148.722
C01188=1169.099,387.890,-83.034,-176.070,9.184,148.721
C01189=1169.102,387.642,-82.999,-176.070,9.182,148.720
C01190=1169.106,387.395,-82.962,-176.070,9.178,148.720
C01191=1169.110,387.148,-82.926,-176.071,9.175,148.719
C01192=1169.114,386.900,-82.891,-176.072,9.172,148.718
C01193=1169.118,386.652,-82.855,-176.072,9.169,148.717
C01194=1169.122,386.405,-82.819,-176.072,9.166,148.717
C01195=1169.125,386.158,-82.783,-176.072,9.162,148.716
C01196=1169.129,385.910,-82.747,-176.073,9.159,148.715
C01197=1169.134,385.663,-82.711,-176.073,9.156,148.714
C01198=1169.137,385.416,-82.676,-176.074,9.153,148.714
C01199=1169.141,385.168,-82.640,-176.075,9.149,148.713
C01200=1169.145,384.920,-82.604,-176.075,9.146,148.712
C01201=1169.149,384.674,-82.568,-176.076,9.143,148.712
C01202=1169.152,384.426,-82.532,-176.076,9.139,148.711
C01203=1169.157,384.178,-82.496,-176.077,9.136,148.710
C01204=1169.161,383.931,-82.461,-176.078,9.133,148.710
C01205=1169.165,383.684,-82.425,-176.078,9.129,148.709
C01206=1169.168,383.436,-82.390,-176.078,9.126,148.708
C01207=1169.173,383.189,-82.354,-176.079,9.123,148.707
C01208=1169.177,382.941,-82.318,-176.080,9.119,148.707
C01209=1169.180,382.694,-82.283,-176.081,9.116,148.706
C01210=1169.184,382.447,-82.247,-176.081,9.112,148.705
C01211=1169.189,382.200,-82.211,-176.082,9.109,148.705
C01212=1169.192,381.952,-82.175,-176.083,9.106,148.704
C01213=1169.196,381.705,-82.140,-176.084,9.102,148.703
C01214=1169.200,381.457,-82.104,-176.085,9.099,148.703
C01215=1169.205,381.210,-82.068,-176.085,9.095,148.702
C01216=1169.208,380.962,-82.033,-176.087,9.092,148.701
C01217=1169.212,380.715,-81.997,-176.087,9.088,148.701
C01218=1169.216,380.467,-81.962,-176.089,9.084,148.700
C01219=1169.219,380.220,-81.926,-176.090,9.081,148.699
C01220=1169.224,379.973,-81.890,-176.090,9.078,148.699
C01221=1169.228,379.725,-81.855,-176.091,9.074,148.698
C01222=1169.232,379.478,-81.819,-176.092,9.071,148.697
C01223=1169.235,379.230,-81.784,-176.094,9.067,148.697
C01224=1169.239,378.983,-81.748,-176.094,9.064,148.696
C01225=1169.243,378.735,-81.714,-176.096,9.060,148.696
C01226=1169.248,378.488,-81.677,-176.097,9.056,148.695
C01227=1169.251,378.240,-81.642,-176.098,9.053,148.694
C01228=1169.255,377.993,-81.606,-176.099,9.049,148.694
C01229=1169.259,377.746,-81.571,-176.100,9.046,148.693
C01230=1169.263,377.498,-81.536,-176.101,9.042,148.692
C01231=1169.267,377.251,-81.500,-176.103,9.038,148.692
C01232=1169.270,377.003,-81.465,-176.104,9.035,148.691
C01233=1169.275,376.757,-81.429,-176.105,9.031,148.690
C01234=1169.279,376.508,-81.394,-176.107,9.027,148.690
C01235=1169.283,376.261,-81.358,-176.108,9.023,148.689
C01236=1169.287,376.013,-81.323,-176.109,9.020,148.689
C01237=1169.291,375.766,-81.288,-176.111,9.016,148.688
C01238=1169.295,375.519,-81.252,-176.112,9.012,148.688
C01239=1169.299,375.271,-81.217,-176.113,9.008,148.687
C01240=1169.302,375.023,-81.182,-176.114,9.005,148.686
C01241=1169.307,374.776,-81.147,-176.116,9.002,148.686
C01242=1169.310,374.529,-81.111,-176.118,8.998,148.685
C01243=1169.314,374.281,-81.076,-176.119,8.994,148.685
C01244=1169.318,374.034,-81.041,-176.121,8.990,148.684
C01245=1169.322,373.786,-81.005,-176.122,8.986,148.684
C01246=1169.326,373.539,-80.970,-176.124,8.982,148.683
C01247=1169.330,373.291,-80.935,-176.126,8.979,148.683
C01248=1169.334,373.044,-80.900,-176.126,8.976,148.682
C01249=1169.338,372.797,-80.864,-176.128,8.972,148.682
C01250=1169.342,372.548,-80.829,-176.130,8.968,148.681
C01251=1169.346,372.302,-80.794,-176.131,8.965,148.681
C01252=1169.350,372.054,-80.759,-176.133,8.961,148.680
C01253=1169.353,371.806,-80.724,-176.135,8.957,148.679
C01254=1169.358,371.559,-80.689,-176.137,8.954,148.679
C01255=1169.362,371.311,-80.654,-176.138,8.950,148.678
C01256=1169.365,371.064,-80.618,-176.140,8.946,148.678
C01257=1169.370,370.817,-80.583,-176.142,8.942,148.678
C01258=1169.374,370.569,-80.548,-176.144,8.938,148.677
C01259=1169.378,370.322,-80.513,-176.146,8.934,148.676
C01260=1169.382,370.074,-80.478,-176.147,8.930,148.676
C01261=1169.386,369.826,-80.443,-176.149,8.927,148.676
C01262=1169.390,369.579,-80.408,-176.151,8.923,148.675
C01263=1169.393,369.332,-80.373,-176.153,8.919,148.675
C01264=1169.397,369.084,-80.339,-176.154,8.916,148.674
C01265=1169.401,368.837,-80.303,-176.156,8.912,148.674
C01266=1169.405,368.589,-80.269,-176.158,8.909,148.673
C01267=1169.409,368.342,-80.233,-176.161,8.904,148.673
C01268=1169.413,368.094,-80.199,-176.162,8.901,148.672
C01269=1169.417,367.846,-80.163,-176.164,8.897,148.672
C01270=1169.421,367.599,-80.129,-176.166,8.893,148.671
C01271=1169.425,367.351,-80.094,-176.168,8.890,148.671
C01272=1169.429,367.104,-80.059,-176.170,8.886,148.671
C01273=1169.433,366.856,-80.024,-176.172,8.882,148.670
C01274=1169.438,366.609,-79.990,-176.174,8.878,148.670
C01275=1169.441,366.361,-79.954,-176.176,8.874,148.669
C01276=1169.446,366.079,-79.914,-176.178,8.870,148.669
C01277=1169.451,365.797,-79.875,-176.181,8.866,148.668
C01278=1169.455,365.515,-79.835,-176.183,8.861,148.668
C01279=1169.459,365.232,-79.796,-176.185,8.858,148.667
C01280=1169.463,364.985,-79.761,-176.188,8.853,148.667
C01281=1169.467,364.737,-79.727,-176.190,8.850,148.667
C01282=1169.471,364.490,-79.692,-176.192,8.846,148.666
C01283=1169.475,364.242,-79.658,-176.193,8.843,148.666
C01284=1169.479,363.995,-79.623,-176.196,8.838,148.666
C01285=1169.483,363.747,-79.588,-176.198,8.835,148.665
C01286=1169.487,363.500,-79.553,-176.200,8.831,148.665
C01287=1169.491,363.252,-79.519,-176.203,8.827,148.664
C01288=1169.495,363.004,-79.485,-176.205,8.824,148.664
C01289=1169.499,362.757,-79.449,-176.207,8.820,148.664
C01290=1169.503,362.510,-79.415,-176.209,8.817,148.663
C01291=1169.507,362.262,-79.380,-176.211,8.812,148.663
C01292=1169.511,362.014,-79.346,-176.214,8.809,148.663
C01293=1169.515,361.766,-79.312,-176.215,8.805,148.662
C01294=1169.519,361.519,-79.277,-176.218,8.801,148.662
C01295=1169.522,361.271,-79.243,-176.220,8.798,148.662
C01296=1169.527,361.024,-79.209,-176.222,8.794,148.661
C01297=1169.531,360.776,-79.174,-176.225,8.790,148.661
C01298=1169.535,360.529,-79.140,-176.227,8.787,148.661
C01299=1169.539,360.280,-79.105,-176.229,8.783,148.660
C01300=1169.543,360.033,-79.071,-176.232,8.779,148.660
C01301=1169.547,359.786,-79.037,-176.234,8.775,148.660
C01302=1169.551,359.538,-79.002,-176.236,8.772,148.659
C01303=1169.555,359.291,-78.968,-176.239,8.768,148.659
C01304=1169.559,359.043,-78.933,-176.241,8.764,148.659
C01305=1169.563,358.795,-78.899,-176.243,8.761,148.658
C01306=1169.567,358.547,-78.864,-176.246,8.757,148.658
C01307=1169.570,358.300,-78.831,-176.248,8.753,148.658
C01308=1169.575,358.053,-78.796,-176.250,8.750,148.658
C01309=1169.578,357.805,-78.762,-176.252,8.746,148.657
C01310=1169.583,357.558,-78.727,-176.255,8.742,148.657
C01311=1169.587,357.310,-78.694,-176.257,8.739,148.657
C01312=1169.591,357.062,-78.659,-176.259,8.736,148.656
C01313=1169.595,356.815,-78.626,-176.262,8.731,148.656
C01314=1169.599,356.566,-78.591,-176.264,8.728,148.656
C01315=1169.603,356.319,-78.557,-176.266,8.725,148.655
C01316=1169.607,356.072,-78.522,-176.269,8.720,148.655
C01317=1169.611,355.824,-78.489,-176.271,8.717,148.655
C01318=1169.615,355.576,-78.455,-176.273,8.714,148.655
C01319=1169.619,355.329,-78.421,-176.275,8.710,148.654
C01320=1169.623,355.081,-78.387,-176.278,8.706,148.654
C01321=1169.627,354.833,-78.353,-176.280,8.702,148.654
C01322=1169.631,354.586,-78.319,-176.282,8.699,148.653
C01323=1169.634,354.338,-78.284,-176.285,8.695,148.653
C01324=1169.639,354.090,-78.251,-176.287,8.691,148.653
C01325=1169.643,353.843,-78.217,-176.289,8.688,148.653
C01326=1169.647,353.595,-78.182,-176.292,8.685,148.652
C01327=1169.651,353.347,-78.149,-176.295,8.681,148.652
C01328=1169.655,353.100,-78.115,-176.296,8.677,148.652
C01329=1169.660,352.852,-78.081,-176.299,8.674,148.651
C01330=1169.663,352.604,-78.047,-176.302,8.670,148.651
C01331=1169.667,352.357,-78.013,-176.304,8.666,148.651
C01332=1169.672,352.109,-77.979,-176.306,8.663,148.651
C01333=1169.676,351.862,-77.945,-176.308,8.660,148.650
C01334=1169.679,351.614,-77.912,-176.311,8.655,148.650
C01335=1169.683,351.366,-77.878,-176.313,8.652,148.650
C01336=1169.688,351.118,-77.844,-176.315,8.649,148.650
C01337=1169.692,350.871,-77.810,-176.318,8.645,148.649
C01338=1169.695,350.623,-77.777,-176.321,8.641,148.649
C01339=1169.700,350.375,-77.742,-176.323,8.638,148.649
C01340=1169.704,350.128,-77.709,-176.325,8.635,148.649
C01341=1169.708,349.881,-77.675,-176.327,8.631,148.648
C01342=1169.711,349.632,-77.642,-176.330,8.627,148.648
C01343=1169.716,349.384,-77.608,-176.332,8.624,148.648
C01344=1169.720,349.137,-77.574,-176.334,8.620,148.648
C01345=1169.724,348.889,-77.541,-176.337,8.617,148.647
C01346=1169.728,348.642,-77.508,-176.340,8.613,148.647
C01347=1169.731,348.394,-77.474,-176.342,8.610,148.647
C01348=1169.736,348.146,-77.440,-176.344,8.606,148.647
C01349=1169.741,347.898,-77.407,-176.346,8.603,148.646
C01350=1169.744,347.651,-77.373,-176.349,8.599,148.646
C01351=1169.748,347.403,-77.340,-176.352,8.596,148.646
C01352=1169.753,347.155,-77.307,-176.354,8.592,148.646
C01353=1169.756,346.908,-77.272,-176.356,8.589,148.646
C01354=1169.760,346.660,-77.239,-176.358,8.585,148.645
C01355=1169.765,346.412,-77.206,-176.361,8.581,148.645
C01356=1169.769,346.164,-77.172,-176.363,8.578,148.645
C01357=1169.773,345.917,-77.139,-176.365,8.575,148.644
C01358=1169.777,345.669,-77.105,-176.368,8.571,148.644
C01359=1169.781,345.422,-77.072,-176.370,8.567,148.644
C01360=1169.785,345.173,-77.039,-176.373,8.564,148.644
C01361=1169.789,344.925,-77.006,-176.375,8.561,148.644
C01362=1169.793,344.678,-76.972,-176.377,8.557,148.643
C01363=1169.797,344.431,-76.938,-176.380,8.553,148.643
C01364=1169.801,344.183,-76.905,-176.382,8.550,148.643
C01365=1169.805,343.935,-76.872,-176.385,8.547,148.643
C01366=1169.809,343.687,-76.839,-176.387,8.543,148.642
C01367=1169.813,343.440,-76.806,-176.390,8.540,148.642
C01368=1169.817,343.192,-76.773,-176.393,8.536,148.642
C01369=1169.822,342.944,-76.740,-176.395,8.533,148.642
C01370=1169.826,342.696,-76.706,-176.397,8.530,148.642
C01371=1169.830,342.449,-76.673,-176.399,8.526,148.642
C01372=1169.834,342.201,-76.640,-176.402,8.522,148.641
C01373=1169.838,341.953,-76.607,-176.405,8.519,148.641
C01374=1169.842,341.705,-76.573,-176.407,8.516,148.641
C01375=1169.846,341.457,-76.540,-176.409,8.512,148.641
C01376=1169.850,341.209,-76.507,-176.411,8.509,148.640
C01377=1169.854,340.962,-76.474,-176.414,8.505,148.640
C01378=1169.858,340.714,-76.441,-176.417,8.502,148.640
C01379=1169.862,340.466,-76.408,-176.419,8.498,148.640
C01380=1169.868,340.187,-76.370,-176.422,8.494,148.639
C01381=1169.872,339.908,-76.333,-176.424,8.491,148.639
C01382=1169.876,339.628,-76.297,-176.427,8.487,148.639
C01383=1169.881,339.348,-76.259,-176.430,8.483,148.639
C01384=1169.885,339.101,-76.226,-176.432,8.480,148.639
C01385=1169.889,338.853,-76.193,-176.435,8.476,148.639
C01386=1169.893,338.605,-76.160,-176.437,8.473,148.638
C01387=1169.897,338.357,-76.127,-176.439,8.470,148.638
C01388=1169.901,338.109,-76.095,-176.443,8.466,148.638
C01389=1169.905,337.862,-76.062,-176.445,8.463,148.638
C01390=1169.909,337.614,-76.028,-176.447,8.459,148.638
C01391=1169.914,337.366,-75.995,-176.450,8.456,148.637
C01392=1169.919,337.119,-75.963,-176.452,8.453,148.637
C01393=1169.922,336.871,-75.931,-176.455,8.449,148.637
C01394=1169.926,336.623,-75.897,-176.457,8.446,148.637
C01395=1169.931,336.375,-75.865,-176.460,8.442,148.637
C01396=1169.935,336.127,-75.832,-176.462,8.439,148.637
C01397=1169.939,335.880,-75.799,-176.464,8.436,148.636
C01398=1169.943,335.632,-75.767,-176.467,8.433,148.636
C01399=1169.947,335.384,-75.734,-176.469,8.428,148.636
C01400=1169.951,335.136,-75.701,-176.472,8.425,148.636
C01401=1169.955,334.888,-75.669,-176.474,8.422,148.636
C01402=1169.959,334.640,-75.636,-176.477,8.419,148.635
C01403=1169.963,334.392,-75.603,-176.479,8.416,148.635
C01404=1169.967,334.144,-75.570,-176.481,8.412,148.635
C01405=1169.971,333.897,-75.538,-176.484,8.409,148.635
C01406=1169.976,333.649,-75.505,-176.487,8.405,148.635
C01407=1169.980,333.401,-75.472,-176.489,8.402,148.635
C01408=1169.984,333.153,-75.440,-176.491,8.399,148.634
C01409=1169.988,332.906,-75.407,-176.494,8.396,148.634
C01410=1169.992,332.657,-75.375,-176.496,8.392,148.634
C01411=1169.996,332.410,-75.342,-176.499,8.389,148.634
C01412=1170.000,332.162,-75.310,-176.501,8.386,148.634
C01413=1170.004,331.914,-75.278,-176.504,8.382,148.634
C01414=1170.008,331.666,-75.245,-176.507,8.379,148.634
C01415=1170.013,331.418,-75.213,-176.509,8.375,148.633
C01416=1170.016,331.171,-75.180,-176.511,8.372,148.633
C01417=1170.021,330.922,-75.148,-176.514,8.369,148.633
C01418=1170.024,330.674,-75.116,-176.516,8.366,148.633
C01419=1170.029,330.427,-75.083,-176.518,8.362,148.633
C01420=1170.033,330.179,-75.051,-176.522,8.359,148.633
C01421=1170.037,329.932,-75.018,-176.524,8.355,148.632
C01422=1170.041,329.683,-74.986,-176.526,8.352,148.632
C01423=1170.045,329.435,-74.954,-176.529,8.349,148.632
C01424=1170.050,329.187,-74.922,-176.531,8.346,148.632
C01425=1170.054,328.940,-74.889,-176.534,8.342,148.632
C01426=1170.058,328.692,-74.857,-176.536,8.339,148.632
C01427=1170.062,328.444,-74.825,-176.539,8.336,148.632
C01428=1170.067,328.196,-74.793,-176.541,8.332,148.631
C01429=1170.070,327.949,-74.760,-176.544,8.329,148.631
C01430=1170.075,327.700,-74.728,-176.546,8.326,148.631
C01431=1170.078,327.452,-74.696,-176.549,8.322,148.631
C01432=1170.083,327.205,-74.664,-176.551,8.319,148.631
C01433=1170.087,326.957,-74.632,-176.554,8.316,148.631
C01434=1170.091,326.709,-74.599,-176.556,8.313,148.631
C01435=1170.095,326.461,-74.567,-176.558,8.310,148.630
C01436=1170.099,326.213,-74.535,-176.561,8.307,148.630
C01437=1170.104,325.965,-74.503,-176.564,8.302,148.630
C01438=1170.107,325.717,-74.471,-176.566,8.299,148.630
C01439=1170.111,325.469,-74.439,-176.569,8.296,148.630
C01440=1170.116,325.221,-74.407,-176.571,8.293,148.630
C01441=1170.120,324.973,-74.375,-176.574,8.290,148.630
C01442=1170.124,324.725,-74.343,-176.576,8.287,148.630
C01443=1170.129,324.478,-74.312,-176.579,8.283,148.629
C01444=1170.132,324.230,-74.280,-176.581,8.280,148.629
C01445=1170.137,323.981,-74.247,-176.584,8.277,148.629
C01446=1170.141,323.734,-74.216,-176.586,8.274,148.629
C01447=1170.145,323.486,-74.184,-176.589,8.270,148.629
C01448=1170.149,323.237,-74.151,-176.591,8.267,148.629
C01449=1170.153,322.989,-74.120,-176.594,8.264,148.629
C01450=1170.157,322.742,-74.088,-176.596,8.260,148.629
C01451=1170.161,322.494,-74.056,-176.599,8.257,148.628
C01452=1170.166,322.246,-74.024,-176.601,8.254,148.628
C01453=1170.170,321.998,-73.992,-176.604,8.251,148.628
C01454=1170.173,321.750,-73.961,-176.606,8.248,148.628
C01455=1170.178,321.503,-73.929,-176.609,8.244,148.628
C01456=1170.182,321.255,-73.897,-176.611,8.241,148.628
C01457=1170.186,321.006,-73.865,-176.614,8.238,148.628
C01458=1170.190,320.759,-73.834,-176.617,8.234,148.628
C01459=1170.194,320.511,-73.802,-176.619,8.231,148.628
C01460=1170.199,320.262,-73.770,-176.622,8.228,148.627
C01461=1170.203,320.015,-73.738,-176.624,8.225,148.627
C01462=1170.207,319.766,-73.707,-176.627,8.222,148.627
C01463=1170.211,319.519,-73.676,-176.629,8.219,148.627
C01464=1170.215,319.271,-73.644,-176.632,8.215,148.627
C01465=1170.219,319.024,-73.612,-176.634,8.212,148.627
C01466=1170.224,318.775,-73.581,-176.637,8.209,148.627
C01467=1170.228,318.527,-73.549,-176.639,8.206,148.627
C01468=1170.232,318.279,-73.517,-176.642,8.203,148.627
C01469=1170.236,318.031,-73.485,-176.644,8.199,148.626
C01470=1170.240,317.783,-73.455,-176.647,8.196,148.626
C01471=1170.244,317.535,-73.423,-176.649,8.193,148.626
C01472=1170.248,317.288,-73.391,-176.652,8.189,148.626
C01473=1170.252,317.039,-73.360,-176.655,8.186,148.626
C01474=1170.257,316.791,-73.328,-176.657,8.183,148.626
C01475=1170.261,316.543,-73.297,-176.660,8.180,148.626
C01476=1170.265,316.295,-73.265,-176.662,8.177,148.626
C01477=1170.269,316.048,-73.234,-176.665,8.173,148.626
C01478=1170.273,315.799,-73.203,-176.667,8.170,148.626
C01479=1170.278,315.552,-73.171,-176.670,8.167,148.626
C01480=1170.282,315.303,-73.140,-176.672,8.164,148.626
C01481=1170.286,315.056,-73.108,-176.675,8.161,148.625
C01482=1170.290,314.807,-73.077,-176.677,8.158,148.625
C01483=1170.294,314.560,-73.046,-176.680,8.155,148.625
C01484=1170.300,314.282,-73.011,-176.683,8.151,148.625
C01485=1170.304,314.006,-72.977,-176.685,8.147,148.625
C01486=1170.309,313.729,-72.941,-176.689,8.144,148.625
C01487=1170.313,313.451,-72.906,-176.691,8.140,148.625
C01488=1170.318,313.203,-72.875,-176.694,8.137,148.625
C01489=1170.322,312.955,-72.844,-176.696,8.134,148.625
C01490=1170.326,312.707,-72.812,-176.699,8.131,148.625
C01491=1170.330,312.460,-72.782,-176.701,8.128,148.625
C01492=1170.334,312.212,-72.750,-176.704,8.125,148.624
C01493=1170.338,311.964,-72.720,-176.706,8.122,148.624
C01494=1170.342,311.715,-72.689,-176.709,8.119,148.624
C01495=1170.347,311.468,-72.657,-176.711,8.116,148.624
C01496=1170.351,311.219,-72.626,-176.714,8.111,148.624
C01497=1170.355,310.971,-72.595,-176.717,8.108,148.624
C01498=1170.360,310.723,-72.564,-176.719,8.105,148.624
C01499=1170.363,310.475,-72.533,-176.722,8.102,148.624
C01500=1170.368,310.227,-72.502,-176.724,8.099,148.624
C01501=1170.372,309.979,-72.472,-176.727,8.096,148.624
C01502=1170.376,309.731,-72.440,-176.730,8.093,148.624
C01503=1170.380,309.483,-72.409,-176.732,8.090,148.623
C01504=1170.384,309.235,-72.378,-176.735,8.087,148.624
C01505=1170.389,308.987,-72.347,-176.737,8.083,148.623
C01506=1170.394,308.739,-72.316,-176.740,8.080,148.623
C01507=1170.398,308.490,-72.285,-176.742,8.077,148.623
C01508=1170.401,308.243,-72.254,-176.745,8.074,148.623
C01509=1170.406,307.995,-72.224,-176.748,8.071,148.623
C01510=1170.410,307.747,-72.192,-176.750,8.068,148.623
C01511=1170.414,307.499,-72.162,-176.753,8.065,148.623
C01512=1170.418,307.251,-72.132,-176.755,8.062,148.623
C01513=1170.422,307.002,-72.100,-176.758,8.059,148.623
C01514=1170.427,306.754,-72.070,-176.760,8.056,148.623
C01515=1170.431,306.506,-72.039,-176.763,8.052,148.623
C01516=1170.435,306.258,-72.008,-176.765,8.049,148.623
C01517=1170.439,306.010,-71.978,-176.768,8.046,148.623
C01518=1170.444,305.762,-71.947,-176.770,8.043,148.623
C01519=1170.448,305.513,-71.916,-176.773,8.040,148.623
C01520=1170.452,305.266,-71.885,-176.775,8.037,148.622
C01521=1170.456,305.018,-71.855,-176.778,8.034,148.622
C01522=1170.461,304.770,-71.824,-176.780,8.031,148.622
C01523=1170.464,304.522,-71.793,-176.783,8.028,148.622
C01524=1170.469,304.274,-71.763,-176.786,8.025,148.622
C01525=1170.474,304.026,-71.732,-176.788,8.021,148.622
C01526=1170.477,303.778,-71.702,-176.791,8.018,148.622
C01527=1170.481,303.529,-71.671,-176.794,8.015,148.622
C01528=1170.486,303.281,-71.640,-176.796,8.012,148.622
C01529=1170.490,303.034,-71.610,-176.799,8.009,148.622
C01530=1170.495,302.785,-71.580,-176.801,8.006,148.622
C01531=1170.499,302.536,-71.548,-176.804,8.003,148.622
C01532=1170.503,302.289,-71.518,-176.806,8.000,148.622
C01533=1170.507,302.041,-71.488,-176.809,7.997,148.622
C01534=1170.511,301.793,-71.457,-176.811,7.994,148.622
C01535=1170.516,301.545,-71.427,-176.814,7.991,148.622
C01536=1170.519,301.296,-71.397,-176.817,7.988,148.622
C01537=1170.524,301.048,-71.366,-176.819,7.984,148.622
C01538=1170.529,300.800,-71.335,-176.822,7.981,148.622
C01539=1170.533,300.552,-71.306,-176.825,7.978,148.622
C01540=1170.537,300.304,-71.275,-176.827,7.975,148.621
C01541=1170.541,300.056,-71.245,-176.830,7.972,148.621
C01542=1170.545,299.808,-71.214,-176.832,7.969,148.621
C01543=1170.550,299.560,-71.184,-176.835,7.966,148.621
C01544=1170.554,299.312,-71.154,-176.837,7.963,148.621
C01545=1170.558,299.064,-71.123,-176.840,7.960,148.621
C01546=1170.563,298.815,-71.093,-176.842,7.957,148.621
C01547=1170.566,298.567,-71.063,-176.845,7.954,148.621
C01548=1170.571,298.318,-71.033,-176.847,7.951,148.621
C01549=1170.575,298.071,-71.003,-176.850,7.948,148.621
C01550=1170.579,297.823,-70.972,-176.852,7.945,148.621
C01551=1170.584,297.575,-70.942,-176.855,7.942,148.621
C01552=1170.588,297.327,-70.912,-176.857,7.939,148.621
C01553=1170.593,297.078,-70.882,-176.860,7.936,148.621
C01554=1170.596,296.830,-70.852,-176.863,7.933,148.621
C01555=1170.601,296.581,-70.822,-176.866,7.930,148.621
C01556=1170.605,296.334,-70.791,-176.868,7.927,148.621
C01557=1170.609,296.086,-70.762,-176.871,7.924,148.621
C01558=1170.613,295.838,-70.731,-176.873,7.921,148.621
C01559=1170.618,295.589,-70.702,-176.876,7.917,148.621
C01560=1170.621,295.342,-70.672,-176.878,7.914,148.621
C01561=1170.626,295.093,-70.641,-176.881,7.911,148.621
C01562=1170.630,294.845,-70.611,-176.884,7.908,148.621
C01563=1170.634,294.597,-70.582,-176.886,7.905,148.621
C01564=1170.639,294.349,-70.552,-176.889,7.902,148.621
C01565=1170.643,294.100,-70.521,-176.892,7.899,148.621
C01566=1170.647,293.852,-70.492,-176.894,7.896,148.621
C01567=1170.651,293.604,-70.461,-176.896,7.894,148.621
C01568=1170.656,293.356,-70.432,-176.899,7.891,148.621
C01569=1170.660,293.107,-70.402,-176.902,7.888,148.621
C01570=1170.664,292.860,-70.372,-176.904,7.885,148.621
C01571=1170.669,292.611,-70.342,-176.907,7.882,148.620
C01572=1170.673,292.363,-70.312,-176.909,7.879,148.621
C01573=1170.677,292.115,-70.283,-176.912,7.876,148.621
C01574=1170.681,291.867,-70.253,-176.915,7.873,148.621
C01575=1170.686,291.618,-70.223,-176.917,7.869,148.620
C01576=1170.690,291.370,-70.193,-176.920,7.866,148.620
C01577=1170.694,291.122,-70.164,-176.923,7.863,148.620
C01578=1170.698,290.874,-70.134,-176.925,7.860,148.620
C01579=1170.702,290.626,-70.104,-176.928,7.857,148.620
C01580=1170.707,290.377,-70.074,-176.930,7.854,148.620
C01581=1170.711,290.129,-70.045,-176.933,7.851,148.620
C01582=1170.715,289.881,-70.015,-176.935,7.849,148.620
C01583=1170.719,289.633,-69.985,-176.938,7.846,148.620
C01584=1170.724,289.385,-69.956,-176.940,7.843,148.620
C01585=1170.728,289.137,-69.926,-176.943,7.840,148.620
C01586=1170.732,288.888,-69.897,-176.946,7.837,148.620
C01587=1170.737,288.640,-69.867,-176.949,7.834,148.620
C01588=1170.742,288.366,-69.835,-176.951,7.831,148.620
C01589=1170.746,288.091,-69.802,-176.955,7.827,148.620
C01590=1170.751,287.815,-69.769,-176.957,7.824,148.620
C01591=1170.756,287.541,-69.736,-176.960,7.821,148.620
C01592=1170.760,287.292,-69.706,-176.962,7.818,148.620
C01593=1170.765,287.045,-69.677,-176.965,7.815,148.620
C01594=1170.769,286.797,-69.648,-176.968,7.812,148.620
C01595=1170.773,286.548,-69.618,-176.971,7.809,148.620
C01596=1170.777,286.300,-69.589,-176.973,7.806,148.620
C01597=1170.782,286.052,-69.560,-176.976,7.803,148.620
C01598=1170.786,285.803,-69.530,-176.978,7.800,148.620
C01599=1170.790,285.555,-69.501,-176.981,7.797,148.620
C01600=1170.794,285.307,-69.471,-176.983,7.795,148.620
C01601=1170.799,285.058,-69.442,-176.986,7.791,148.620
C01602=1170.803,284.810,-69.413,-176.988,7.788,148.620
C01603=1170.808,284.562,-69.384,-176.991,7.785,148.620
C01604=1170.812,284.314,-69.354,-176.994,7.782,148.620
C01605=1170.816,284.066,-69.325,-176.997,7.779,148.620
C01606=1170.820,283.817,-69.296,-176.999,7.776,148.620
C01607=1170.824,283.569,-69.266,-177.002,7.773,148.620
C01608=1170.829,283.320,-69.237,-177.004,7.770,148.620
C01609=1170.834,283.073,-69.208,-177.006,7.768,148.620
C01610=1170.838,282.824,-69.179,-177.009,7.765,148.620
C01611=1170.842,282.576,-69.149,-177.012,7.762,148.620
C01612=1170.846,282.328,-69.120,-177.015,7.759,148.621
C01613=1170.850,282.079,-69.092,-177.017,7.756,148.621
C01614=1170.855,281.832,-69.063,-177.020,7.753,148.621
C01615=1170.859,281.583,-69.033,-177.022,7.750,148.620
C01616=1170.863,281.335,-69.004,-177.025,7.747,148.620
C01617=1170.867,281.086,-68.975,-177.027,7.745,148.621
C01618=1170.872,280.838,-68.946,-177.030,7.742,148.621
C01619=1170.877,280.590,-68.917,-177.033,7.739,148.621
C01620=1170.881,280.342,-68.888,-177.036,7.736,148.621
C01621=1170.884,280.094,-68.859,-177.038,7.733,148.621
C01622=1170.889,279.845,-68.830,-177.041,7.730,148.621
C01623=1170.894,279.597,-68.801,-177.043,7.727,148.621
C01624=1170.898,279.349,-68.772,-177.046,7.724,148.621
C01625=1170.902,279.100,-68.743,-177.048,7.721,148.621
C01626=1170.906,278.852,-68.714,-177.051,7.718,148.621
C01627=1170.911,278.604,-68.686,-177.054,7.715,148.621
C01628=1170.915,278.356,-68.656,-177.057,7.712,148.621
C01629=1170.919,278.107,-68.627,-177.059,7.709,148.621
C01630=1170.923,277.859,-68.599,-177.062,7.707,148.621
C01631=1170.928,277.611,-68.570,-177.064,7.704,148.621
C01632=1170.932,277.362,-68.541,-177.067,7.701,148.621
C01633=1170.937,277.113,-68.512,-177.069,7.698,148.621
C01634=1170.941,276.866,-68.484,-177.072,7.695,148.621
C01635=1170.945,276.617,-68.455,-177.075,7.692,148.621
C01636=1170.949,276.369,-68.425,-177.077,7.689,148.621
C01637=1170.953,276.120,-68.397,-177.080,7.686,148.621
C01638=1170.958,275.873,-68.368,-177.082,7.684,148.621
C01639=1170.962,275.624,-68.339,-177.085,7.681,148.621
C01640=1170.966,275.375,-68.311,-177.088,7.678,148.621
C01641=1170.971,275.128,-68.282,-177.091,7.675,148.621
C01642=1170.975,274.879,-68.253,-177.093,7.672,148.621
C01643=1170.979,274.631,-68.225,-177.096,7.669,148.621
C01644=1170.984,274.383,-68.196,-177.098,7.667,148.621
C01645=1170.988,274.134,-68.167,-177.101,7.664,148.621
C01646=1170.993,273.887,-68.139,-177.104,7.661,148.622
C01647=1170.997,273.638,-68.110,-177.107,7.658,148.622
C01648=1171.001,273.389,-68.081,-177.109,7.655,148.621
C01649=1171.006,273.141,-68.054,-177.112,7.652,148.621
C01650=1171.010,272.893,-68.024,-177.114,7.650,148.622
C01651=1171.014,272.644,-67.996,-177.116,7.647,148.622
C01652=1171.019,272.396,-67.968,-177.119,7.644,148.622
C01653=1171.023,272.147,-67.940,-177.122,7.641,148.622
C01654=1171.027,271.900,-67.910,-177.125,7.638,148.622
C01655=1171.032,271.651,-67.882,-177.127,7.636,148.622
C01656=1171.036,271.402,-67.854,-177.130,7.633,148.622
C01657=1171.041,271.154,-67.825,-177.132,7.630,148.622
C01658=1171.044,270.906,-67.797,-177.135,7.627,148.622
C01659=1171.050,270.657,-67.769,-177.138,7.624,148.622
C01660=1171.053,270.409,-67.740,-177.141,7.621,148.622
C01661=1171.058,270.161,-67.711,-177.143,7.619,148.622
C01662=1171.062,269.913,-67.683,-177.146,7.616,148.622
C01663=1171.066,269.664,-67.655,-177.148,7.613,148.622
C01664=1171.071,269.416,-67.627,-177.151,7.610,148.622
C01665=1171.075,269.167,-67.598,-177.154,7.607,148.622
C01666=1171.080,268.919,-67.570,-177.156,7.605,148.622
C01667=1171.083,268.671,-67.542,-177.159,7.602,148.622
C01668=1171.088,268.422,-67.514,-177.161,7.599,148.623
C01669=1171.092,268.174,-67.486,-177.164,7.596,148.623
C01670=1171.097,267.926,-67.457,-177.167,7.593,148.623
C01671=1171.101,267.677,-67.429,-177.169,7.591,148.623
C01672=1171.106,267.429,-67.401,-177.172,7.588,148.623
C01673=1171.110,267.180,-67.373,-177.175,7.585,148.623
C01674=1171.114,266.932,-67.345,-177.177,7.582,148.623
C01675=1171.119,266.684,-67.316,-177.180,7.580,148.623
C01676=1171.123,266.436,-67.288,-177.182,7.577,148.623
C01677=1171.127,266.187,-67.260,-177.185,7.574,148.623
C01678=1171.132,265.939,-67.232,-177.188,7.571,148.623
C01679=1171.136,265.690,-67.204,-177.191,7.568,148.623
C01680=1171.141,265.442,-67.176,-177.193,7.566,148.623
C01681=1171.145,265.194,-67.148,-177.195,7.563,148.623
C01682=1171.149,264.945,-67.120,-177.198,7.560,148.623
C01683=1171.154,264.697,-67.092,-177.201,7.557,148.623
C01684=1171.158,264.448,-67.064,-177.204,7.555,148.624
C01685=1171.162,264.200,-67.036,-177.206,7.552,148.624
C01686=1171.166,263.951,-67.008,-177.209,7.549,148.624
C01687=1171.171,263.703,-66.980,-177.212,7.546,148.624
C01688=1171.175,263.454,-66.952,-177.215,7.543,148.624
C01689=1171.179,263.207,-66.924,-177.217,7.541,148.624
C01690=1171.184,262.958,-66.897,-177.220,7.538,148.624
C01691=1171.189,262.709,-66.868,-177.222,7.535,148.624
C01692=1171.194,262.437,-66.838,-177.225,7.532,148.624
C01693=1171.199,262.163,-66.807,-177.228,7.529,148.624
C01694=1171.203,261.890,-66.777,-177.231,7.526,148.624
C01695=1171.208,261.617,-66.746,-177.234,7.523,148.625
C01696=1171.212,261.369,-66.718,-177.236,7.521,148.625
C01697=1171.217,261.121,-66.690,-177.239,7.518,148.625
C01698=1171.221,260.872,-66.663,-177.242,7.515,148.625
C01699=1171.225,260.624,-66.635,-177.244,7.512,148.625
C01700=1171.230,260.376,-66.607,-177.247,7.509,148.625
C01701=1171.234,260.126,-66.579,-177.250,7.507,148.625
C01702=1171.238,259.879,-66.552,-177.252,7.504,148.625
C01703=1171.243,259.629,-66.524,-177.255,7.501,148.625
C01704=1171.247,259.381,-66.496,-177.257,7.498,148.625
C01705=1171.252,259.133,-66.469,-177.261,7.496,148.625
C01706=1171.255,258.884,-66.441,-177.263,7.493,148.625
C01707=1171.260,258.637,-66.413,-177.265,7.491,148.626
C01708=1171.265,258.388,-66.386,-177.268,7.488,148.626
C01709=1171.269,258.140,-66.358,-177.271,7.485,148.626
C01710=1171.273,257.891,-66.331,-177.273,7.483,148.626
C01711=1171.278,257.642,-66.304,-177.276,7.480,148.626
C01712=1171.282,257.394,-66.276,-177.279,7.477,148.626
C01713=1171.287,257.145,-66.248,-177.282,7.474,148.626
C01714=1171.291,256.897,-66.221,-177.284,7.472,148.626
C01715=1171.296,256.649,-66.193,-177.287,7.469,148.626
C01716=1171.299,256.400,-66.165,-177.290,7.466,148.626
C01717=1171.304,256.152,-66.138,-177.292,7.464,148.626
C01718=1171.309,255.903,-66.111,-177.294,7.461,148.626
C01719=1171.313,255.655,-66.083,-177.297,7.458,148.627
C01720=1171.317,255.406,-66.056,-177.300,7.455,148.627
C01721=1171.322,255.158,-66.029,-177.303,7.453,148.627
C01722=1171.326,254.910,-66.001,-177.305,7.450,148.627
C01723=1171.331,254.661,-65.974,-177.308,7.447,148.627
C01724=1171.335,254.412,-65.947,-177.310,7.445,148.627
C01725=1171.339,254.164,-65.919,-177.313,7.442,148.627
C01726=1171.344,253.916,-65.892,-177.316,7.439,148.627
C01727=1171.348,253.667,-65.865,-177.319,7.437,148.628
C01728=1171.353,253.419,-65.838,-177.321,7.434,148.628
C01729=1171.357,253.170,-65.810,-177.324,7.431,148.628
C01730=1171.361,252.922,-65.783,-177.327,7.428,148.628
C01731=1171.365,252.673,-65.756,-177.329,7.426,148.628
C01732=1171.370,252.425,-65.729,-177.332,7.423,148.628
C01733=1171.374,252.177,-65.701,-177.335,7.421,148.628
C01734=1171.378,251.928,-65.674,-177.337,7.419,148.628
C01735=1171.383,251.679,-65.647,-177.340,7.416,148.628
C01736=1171.388,251.431,-65.620,-177.343,7.413,148.628
C01737=1171.392,251.182,-65.593,-177.345,7.411,148.628
C01738=1171.397,250.934,-65.566,-177.348,7.408,148.629
C01739=1171.401,250.686,-65.539,-177.351,7.405,148.629
C01740=1171.405,250.436,-65.512,-177.353,7.402,148.629
C01741=1171.409,250.189,-65.484,-177.356,7.400,148.629
C01742=1171.414,249.940,-65.457,-177.358,7.397,148.629
C01743=1171.419,249.692,-65.430,-177.362,7.394,148.629
C01744=1171.423,249.443,-65.403,-177.364,7.392,148.629
C01745=1171.427,249.195,-65.376,-177.367,7.389,148.629
C01746=1171.432,248.946,-65.349,-177.369,7.386,148.630
C01747=1171.436,248.697,-65.322,-177.371,7.384,148.630
C01748=1171.441,248.449,-65.295,-177.375,7.381,148.630
C01749=1171.445,248.201,-65.268,-177.377,7.378,148.630
C01750=1171.449,247.952,-65.241,-177.380,7.376,148.630
C01751=1171.454,247.704,-65.214,-177.382,7.373,148.630
C01752=1171.459,247.455,-65.187,-177.386,7.371,148.630
C01753=1171.462,247.207,-65.161,-177.388,7.369,148.631
C01754=1171.467,246.958,-65.133,-177.391,7.366,148.631
C01755=1171.472,246.709,-65.107,-177.393,7.363,148.631
C01756=1171.476,246.461,-65.081,-177.396,7.361,148.631
C01757=1171.481,246.213,-65.054,-177.399,7.358,148.631
C01758=1171.485,245.963,-65.026,-177.401,7.356,148.631
C01759=1171.489,245.715,-65.000,-177.404,7.353,148.631
C01760=1171.493,245.467,-64.973,-177.407,7.350,148.632
C01761=1171.498,245.218,-64.946,-177.409,7.348,148.632
C01762=1171.502,244.969,-64.920,-177.412,7.345,148.632
C01763=1171.507,244.721,-64.893,-177.415,7.342,148.632
C01764=1171.511,244.472,-64.866,-177.417,7.340,148.632
C01765=1171.515,244.224,-64.839,-177.420,7.337,148.632
C01766=1171.520,243.976,-64.812,-177.423,7.334,148.632
C01767=1171.525,243.727,-64.786,-177.425,7.332,148.632
C01768=1171.529,243.478,-64.759,-177.428,7.330,148.633
C01769=1171.534,243.230,-64.732,-177.430,7.327,148.633
C01770=1171.537,242.982,-64.706,-177.433,7.325,148.633
C01771=1171.542,242.733,-64.679,-177.436,7.322,148.633
C01772=1171.546,242.484,-64.653,-177.438,7.320,148.633
C01773=1171.551,242.236,-64.626,-177.441,7.317,148.633
C01774=1171.556,241.987,-64.600,-177.444,7.314,148.633
C01775=1171.560,241.739,-64.573,-177.447,7.312,148.634
C01776=1171.565,241.490,-64.546,-177.449,7.309,148.634
C01777=1171.569,241.241,-64.520,-177.452,7.307,148.634
C01778=1171.573,240.993,-64.493,-177.455,7.304,148.634
C01779=1171.578,240.744,-64.468,-177.457,7.301,148.634
C01780=1171.582,240.496,-64.440,-177.460,7.299,148.634
C01781=1171.586,240.247,-64.414,-177.463,7.297,148.635
C01782=1171.592,239.999,-64.388,-177.465,7.294,148.635
C01783=1171.596,239.751,-64.362,-177.468,7.292,148.635
C01784=1171.601,239.502,-64.335,-177.471,7.289,148.635
C01785=1171.605,239.253,-64.309,-177.473,7.287,148.635
C01786=1171.610,239.004,-64.282,-177.476,7.284,148.635
C01787=1171.613,238.756,-64.256,-177.478,7.282,148.635
C01788=1171.618,238.507,-64.230,-177.481,7.279,148.636
C01789=1171.622,238.259,-64.203,-177.484,7.276,148.636
C01790=1171.627,238.010,-64.177,-177.486,7.274,148.636
C01791=1171.631,237.762,-64.150,-177.490,7.271,148.636
C01792=1171.635,237.513,-64.125,-177.492,7.269,148.636
C01793=1171.640,237.265,-64.098,-177.495,7.267,148.636
C01794=1171.645,237.016,-64.072,-177.498,7.264,148.636
C01795=1171.649,236.767,-64.046,-177.500,7.261,148.637
C01796=1171.654,236.496,-64.017,-177.503,7.259,148.637
C01797=1171.659,236.224,-63.989,-177.506,7.256,148.637
C01798=1171.663,235.953,-63.960,-177.509,7.253,148.637
C01799=1171.669,235.680,-63.932,-177.512,7.250,148.637
C01800=1171.673,235.432,-63.905,-177.515,7.248,148.638
C01801=1171.677,235.183,-63.879,-177.517,7.246,148.638
C01802=1171.683,234.935,-63.853,-177.519,7.243,148.638
C01803=1171.686,234.687,-63.827,-177.523,7.241,148.638
C01804=1171.691,234.438,-63.801,-177.525,7.238,148.638
C01805=1171.696,234.189,-63.775,-177.528,7.236,148.638
C01806=1171.700,233.941,-63.748,-177.531,7.233,148.639
C01807=1171.704,233.693,-63.723,-177.533,7.231,148.639
C01808=1171.709,233.444,-63.697,-177.536,7.228,148.639
C01809=1171.714,233.195,-63.671,-177.538,7.226,148.639
